// NETWORK 10
SIREN_BEACONS(ESTOP_ACTIVE := GVL_Alarms.EMERGENCY_STOP_COMMON, ERRORS_ACTIVE := APP_WARNINGS_ERRORS.ERRORS_ACTIVE, WARNINGS_ACTIVE := APP_WARNINGS_ERRORS.WARNINGS_ACTIVE);

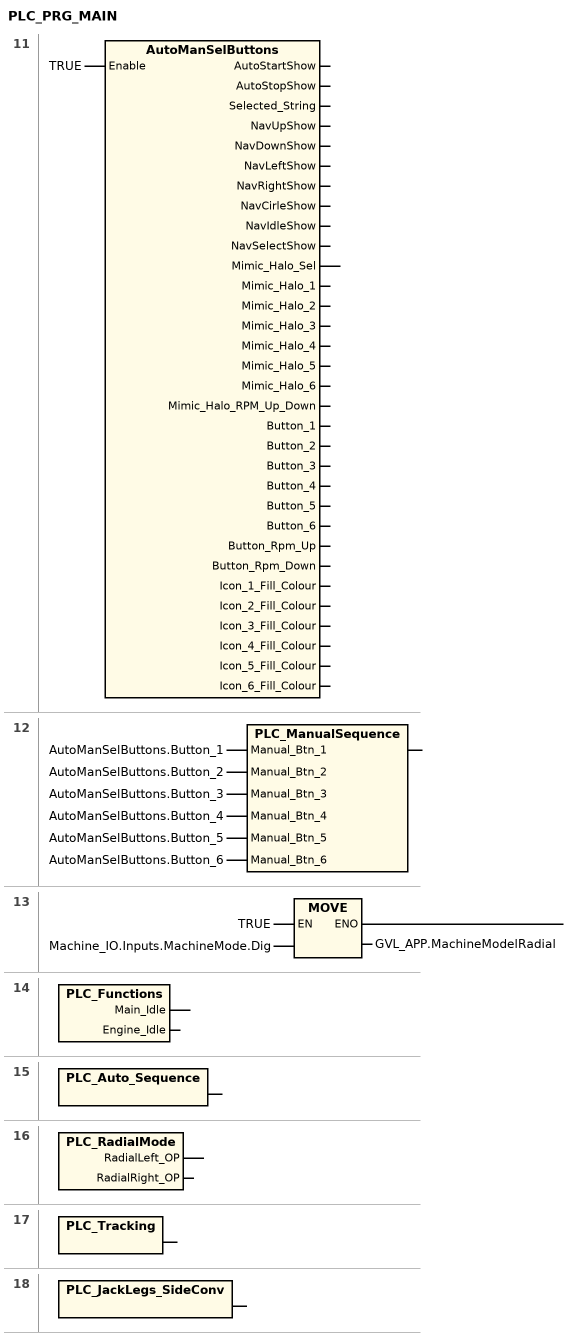
// NETWORK 11
AutoManSelButtons(Enable := TRUE);

// NETWORK 12
PLC_ManualSequence(Manual_Btn_1 := AutoManSelButtons.Button_1, Manual_Btn_2 := AutoManSelButtons.Button_2, Manual_Btn_3 := AutoManSelButtons.Button_3, Manual_Btn_4 := AutoManSelButtons.Button_4, Manual_Btn_5 := AutoManSelButtons.Button_5, Manual_Btn_6 := AutoManSelButtons.Button_6);

// NETWORK 13
GVL_APP.MachineModelRadial := Machine_IO.Inputs.MachineMode.Dig;

// NETWORK 14
PLC_Functions();

// NETWORK 15
PLC_Auto_Sequence();

// NETWORK 16
PLC_RadialMode();

// NETWORK 17
PLC_Tracking();

// NETWORK 18
PLC_JackLegs_SideConv();

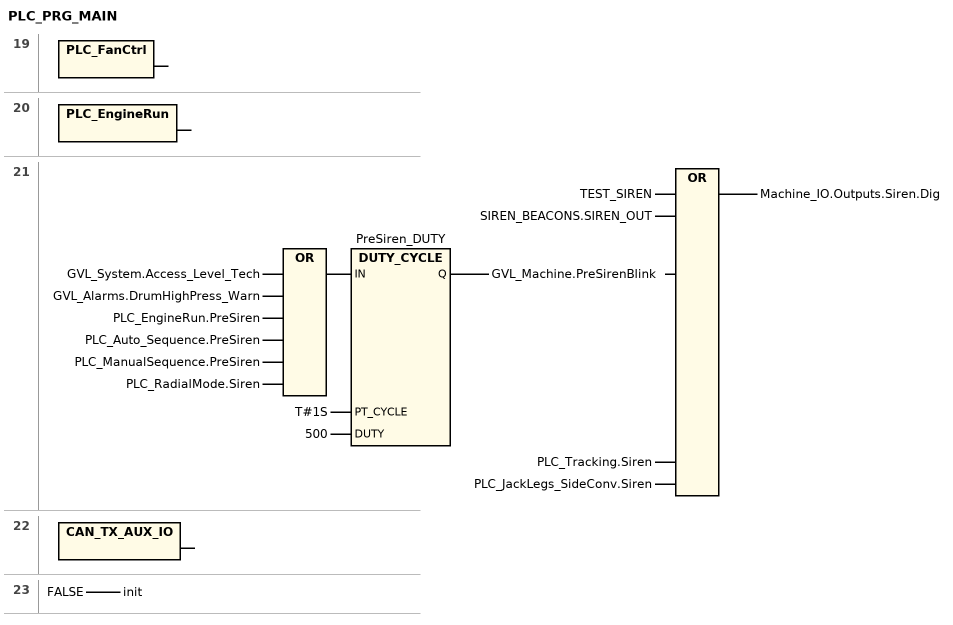
// NETWORK 19
PLC_FanCtrl();

// NETWORK 20
PLC_EngineRun();

// NETWORK 21
PreSiren_DUTY(
    IN := GVL_System.Access_Level_Tech OR GVL_Alarms.DrumHighPress_Warn OR PLC_EngineRun.PreSiren OR PLC_Auto_Sequence.PreSiren OR PLC_ManualSequence.PreSiren OR PLC_RadialMode.Siren,
    PT_CYCLE := T#1S,
    DUTY := 500); // DUTY_CYCLE
GVL_Machine.PreSirenBlink := PreSiren_DUTY.Q;
Machine_IO.Outputs.Siren.Dig := TEST_SIREN OR SIREN_BEACONS.SIREN_OUT OR PreSiren_DUTY.Q OR PLC_Tracking.Siren OR PLC_JackLegs_SideConv.Siren;

// NETWORK 22
CAN_TX_AUX_IO();

// NETWORK 23
init := FALSE;

END_PROGRAM

// Device/Application/App_PLC/PLC_SIM_MAIN
PROGRAM PLC_SIM_MAIN
VAR
END_VAR

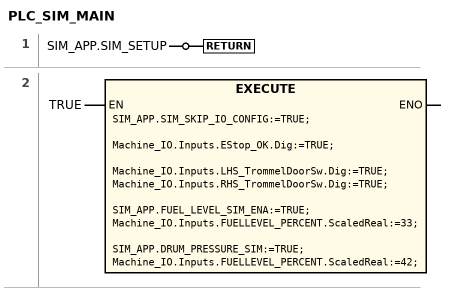
// NETWORK 1
IF NOT SIM_APP.SIM_SETUP THEN RETURN; END_IF

// NETWORK 2
SIM_APP.SIM_SKIP_IO_CONFIG:=TRUE;

Machine_IO.Inputs.EStop_OK.Dig:=TRUE;

Machine_IO.Inputs.LHS_TrommelDoorSw.Dig:=TRUE;
Machine_IO.Inputs.RHS_TrommelDoorSw.Dig:=TRUE;

SIM_APP.FUEL_LEVEL_SIM_ENA:=TRUE;
Machine_IO.Inputs.FUELLEVEL_PERCENT.ScaledReal:=33;

SIM_APP.DRUM_PRESSURE_SIM:=TRUE;
Machine_IO.Inputs.FUELLEVEL_PERCENT.ScaledReal:=42;

END_PROGRAM

// Device/Application/App_Common/System/PLC_COMMON
PROGRAM PLC_COMMON
VAR
	INIT: BOOL := TRUE;

	MAIN_HMI_Version_Info: PLC_Version_Unpack_FB;
	Version_Refresh_TON: TON;
	CHASSIS_PLC_Version_Info: SLL_IFM_Version.PLC_Version_Unpack_FB;
	
	PC_SIMULATION_MODE: INT;
	SIM_PRIME_PULSE_TON: TON;
	SIM_CAS_PRIME_PULSE_TON: TON;
	Get_Task_Info_FB: Get_Task_Info;
	TaskInfo: HMI_TASKS_INFO_STRUCT;
	SetKeyLED_FB: ifmDevice.SetKeyLED;
	
	BOOT_PIN_CODE_ENTERED: LWORD;
	BOOT_PIN_CODE_FIXED: LWORD:=2103;
	BOOT_PIN_CODE_VALID: BOOL;
	BOOT_INTO_RECOVERY: BOOL;
	BOOT_INTO_SETUP: BOOL;
	
 	BootIntoRecovery_FB: ifmDevice.BootIntoRecovery;
// 	BootIntoSetup_FB: ifmDevice.BootIntoSetup;	
 	PrintScreen_FB: ifmDevice.PrintScreen;
 	LoadSplashScreen_FB: ifmDevice.LoadSplashScreen;	
 	PrintScreenPath: STRING := '/home/cds-apps/PlcLogic/';
	SLASH_LOGO_SET: BOOL;
	HideSplashScreen_FB: ifmDevice.HideSplashScreen;
	Load_Splash_TEST: BOOL;
END_VAR

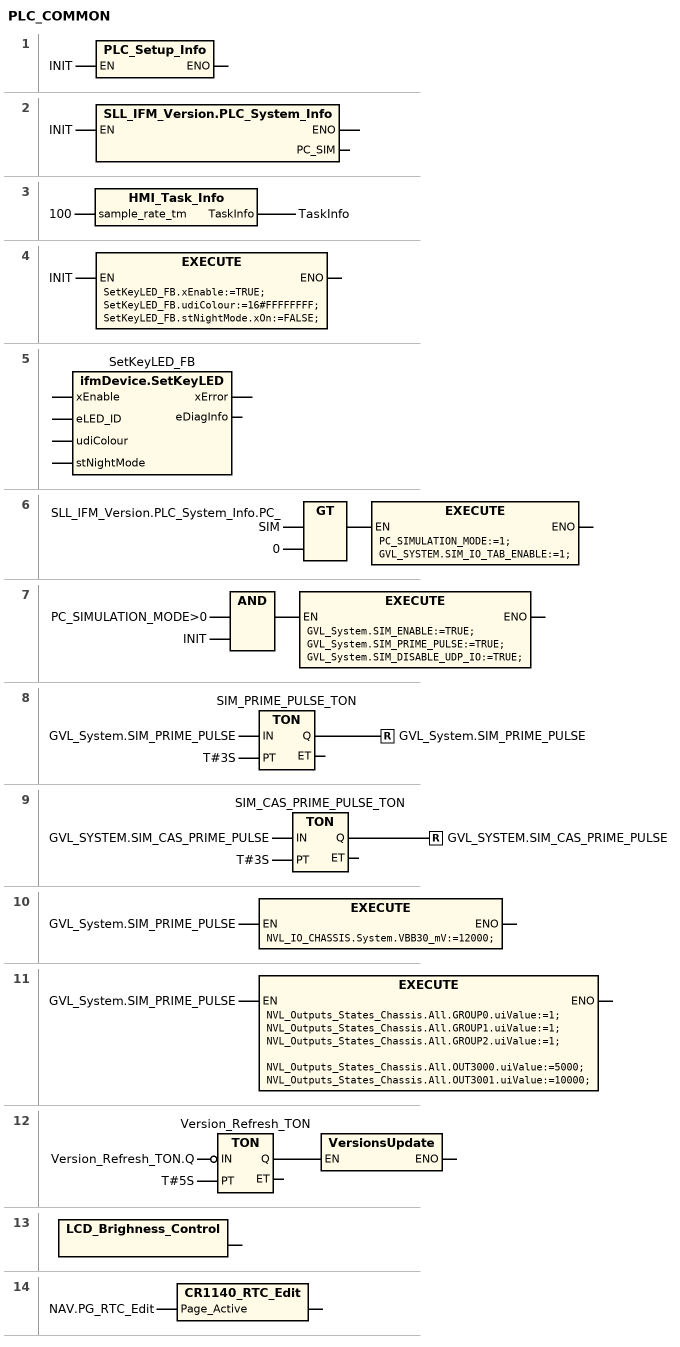
// NETWORK 1
IF INIT THEN PLC_Setup_Info(); END_IF

// NETWORK 2
IF INIT THEN SLL_IFM_Version.PLC_System_Info(); END_IF

// NETWORK 3
HMI_Task_Info(sample_rate_tm := 100);
TaskInfo := HMI_Task_Info.TaskInfo;

// NETWORK 4
IF INIT THEN
    SetKeyLED_FB.xEnable:=TRUE;
    SetKeyLED_FB.udiColour:=16#FFFFFFFF;
    SetKeyLED_FB.stNightMode.xOn:=FALSE;
END_IF

// NETWORK 5
SetKeyLED_FB(); // ifmDevice.SetKeyLED

// NETWORK 6
IF SLL_IFM_Version.PLC_System_Info.PC_SIM > 0 THEN
    PC_SIMULATION_MODE:=1;
    GVL_SYSTEM.SIM_IO_TAB_ENABLE:=1;
END_IF

// NETWORK 7
IF (PC_SIMULATION_MODE>0) AND INIT THEN
    GVL_System.SIM_ENABLE:=TRUE;
    GVL_System.SIM_PRIME_PULSE:=TRUE;
    GVL_System.SIM_DISABLE_UDP_IO:=TRUE;
END_IF

// NETWORK 8
SIM_PRIME_PULSE_TON(IN := GVL_System.SIM_PRIME_PULSE, PT := T#3S); // TON
GVL_System.SIM_PRIME_PULSE R= SIM_PRIME_PULSE_TON.Q;

// NETWORK 9
SIM_CAS_PRIME_PULSE_TON(IN := GVL_SYSTEM.SIM_CAS_PRIME_PULSE, PT := T#3S); // TON
GVL_SYSTEM.SIM_CAS_PRIME_PULSE R= SIM_CAS_PRIME_PULSE_TON.Q;

// NETWORK 10
IF GVL_System.SIM_PRIME_PULSE THEN NVL_IO_CHASSIS.System.VBB30_mV:=12000; END_IF

// NETWORK 11
IF GVL_System.SIM_PRIME_PULSE THEN
    NVL_Outputs_States_Chassis.All.GROUP0.uiValue:=1;
    NVL_Outputs_States_Chassis.All.GROUP1.uiValue:=1;
    NVL_Outputs_States_Chassis.All.GROUP2.uiValue:=1;
    
    NVL_Outputs_States_Chassis.All.OUT3000.uiValue:=5000;
    NVL_Outputs_States_Chassis.All.OUT3001.uiValue:=10000;
END_IF

// NETWORK 12
Version_Refresh_TON(IN := NOT Version_Refresh_TON.Q, PT := T#5S); // TON
IF Version_Refresh_TON.Q THEN VersionsUpdate(); END_IF

// NETWORK 13
LCD_Brighness_Control();

// NETWORK 14
CR1140_RTC_Edit(Page_Active := NAV.PG_RTC_Edit);

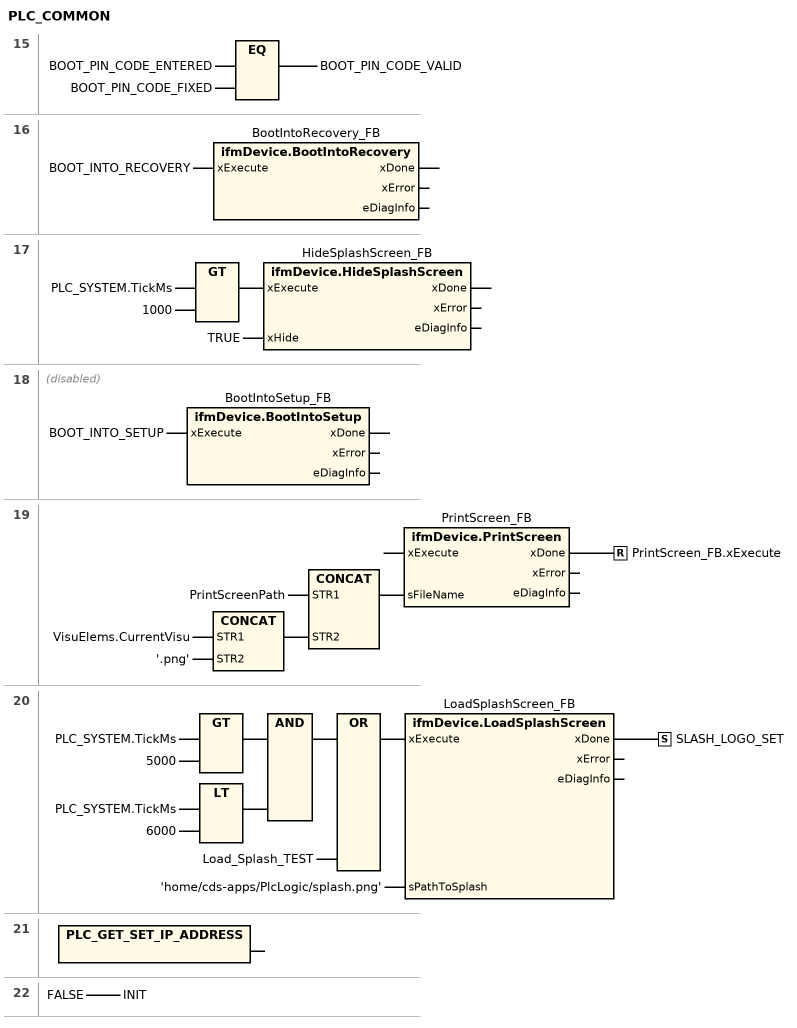
// NETWORK 15
BOOT_PIN_CODE_VALID := BOOT_PIN_CODE_ENTERED = BOOT_PIN_CODE_FIXED;

// NETWORK 16
BootIntoRecovery_FB(xExecute := BOOT_INTO_RECOVERY); // ifmDevice.BootIntoRecovery

// NETWORK 17
HideSplashScreen_FB(xExecute := PLC_SYSTEM.TickMs > 1000, xHide := TRUE); // ifmDevice.HideSplashScreen

// NETWORK 18 (disabled)
// BootIntoSetup_FB(xExecute := BOOT_INTO_SETUP); // ifmDevice.BootIntoSetup

// NETWORK 19
PrintScreen_FB(sFileName := CONCAT(STR1 := PrintScreenPath, STR2 := CONCAT(STR1 := VisuElems.CurrentVisu, STR2 := '.png'))); // ifmDevice.PrintScreen
PrintScreen_FB.xExecute R= PrintScreen_FB.xDone;

// NETWORK 20
LoadSplashScreen_FB(xExecute := PLC_SYSTEM.TickMs > 5000 AND PLC_SYSTEM.TickMs < 6000 OR Load_Splash_TEST, sPathToSplash := 'home/cds-apps/PlcLogic/splash.png'); // ifmDevice.LoadSplashScreen
SLASH_LOGO_SET S= LoadSplashScreen_FB.xDone;

// NETWORK 21
PLC_GET_SET_IP_ADDRESS();

// NETWORK 22
INIT := FALSE;

METHOD VersionsUpdate
VAR_INPUT
END_VAR
VAR
END_VAR
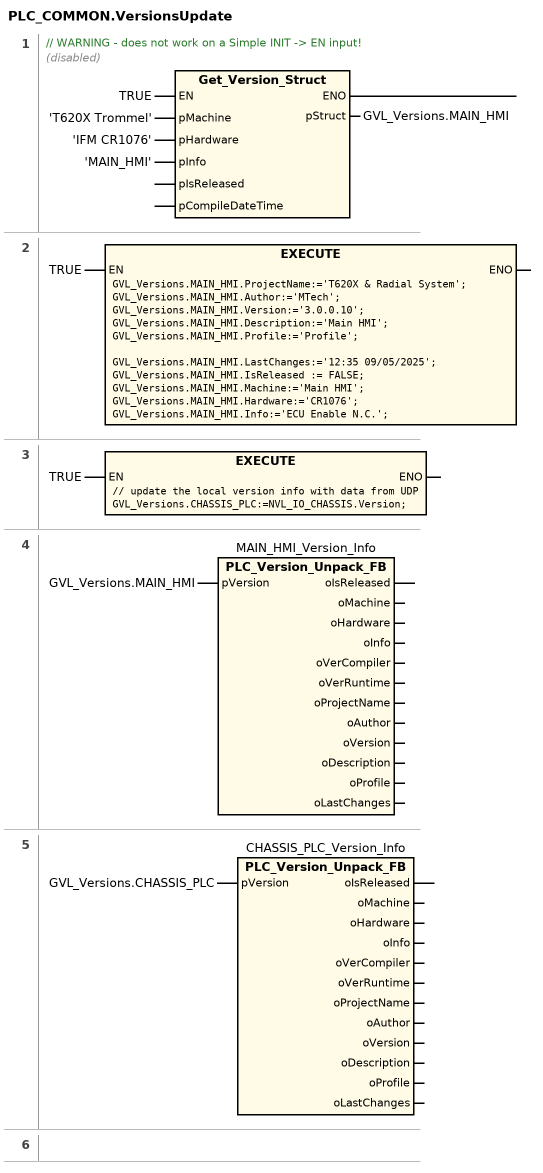
// NETWORK 1 (disabled)
// // WARNING - does not work on a Simple INIT -> EN input!
// Get_Version_Struct(pMachine := 'T620X Trommel', pHardware := 'IFM CR1076', pInfo := 'MAIN_HMI', pStruct => GVL_Versions.MAIN_HMI);

// NETWORK 2
GVL_Versions.MAIN_HMI.ProjectName:='T620X & Radial System';				
GVL_Versions.MAIN_HMI.Author:='MTech';
GVL_Versions.MAIN_HMI.Version:='3.0.0.10';
GVL_Versions.MAIN_HMI.Description:='Main HMI';
GVL_Versions.MAIN_HMI.Profile:='Profile';

GVL_Versions.MAIN_HMI.LastChanges:='12:35 09/05/2025';
GVL_Versions.MAIN_HMI.IsReleased := FALSE;
GVL_Versions.MAIN_HMI.Machine:='Main HMI';
GVL_Versions.MAIN_HMI.Hardware:='CR1076';
GVL_Versions.MAIN_HMI.Info:='ECU Enable N.C.';

// NETWORK 3
// update the local version info with data from UDP
GVL_Versions.CHASSIS_PLC:=NVL_IO_CHASSIS.Version;

// NETWORK 4
MAIN_HMI_Version_Info(pVersion := GVL_Versions.MAIN_HMI); // PLC_Version_Unpack_FB

// NETWORK 5
CHASSIS_PLC_Version_Info(pVersion := GVL_Versions.CHASSIS_PLC); // PLC_Version_Unpack_FB

// NETWORK 6
END_METHOD

END_PROGRAM

// Device/Application/App_Common/System/PLC_Setup_Info
PROGRAM PLC_Setup_Info
VAR
	INIT: BOOL:=TRUE;
END_VAR

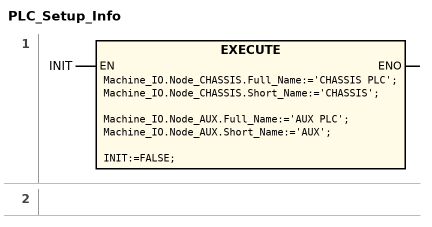
// NETWORK 1
IF INIT THEN
    Machine_IO.Node_CHASSIS.Full_Name:='CHASSIS PLC';
    Machine_IO.Node_CHASSIS.Short_Name:='CHASSIS';
    
    Machine_IO.Node_AUX.Full_Name:='AUX PLC';
    Machine_IO.Node_AUX.Short_Name:='AUX';
    
    INIT:=FALSE;
END_IF

// NETWORK 2

END_PROGRAM

// Device/Application/LIBS/HMI/HMI_Task_Info
PROGRAM HMI_Task_Info
VAR_INPUT
	sample_rate_tm:DWORD:=500;
END_VAR
VAR
	x: INT;
    hTasks:	ARRAY [0..19] OF SysTypes.RTS_IEC_HANDLE;	
    iecResult:	ARRAY [0..19] OF SysTypes.RTS_IEC_RESULT;
    sAppName:	STRING := 'Application';
    pIecInfo:	POINTER TO CmpIecTask.Task_Info2;
	last_sample_ms: DWORD;
	diff_ms: DWORD;
	finished: BOOL := FALSE;
	CpuLoadTemp: REAL;
END_VAR

VAR_OUTPUT
	TaskInfo: HMI_TASKS_INFO_STRUCT;
	CpuLoad:REAL;
END_VAR

diff_ms := SysTimeGetMs() - last_sample_ms;

IF diff_ms < sample_rate_tm THEN
	RETURN;
END_IF

x:=0;
finished:=FALSE;
CpuLoadTemp:=0;

WHILE finished = FALSE DO
	IF x = 0 THEN
		hTasks[x] := CmpIecTask.IecTaskGetFirst(pszAppName := ADR(sAppName), pResult := ADR(iecResult));
	ELSE
		hTasks[x] := IecTaskGetNext(pszAppName := ADR(sAppName), hPrevIecTask := hTasks[x-1], pResult := ADR(iecResult));
	END_IF

	IF ((hTasks[x] <> SysTypes.RTS_INVALID_HANDLE) AND (iecResult[x] = CmpErrors.Errors.ERR_OK)) THEN
		pIecInfo := CmpIecTask.IecTaskGetInfo3(hIecTask := hTasks[x],pResult := ADR(iecResult[x]));
		TaskInfo.Tasks[x].dwIntervalTask := pIecInfo^.dwInterval;
		TaskInfo.Tasks[x].dwCycleTimeTask := pIecInfo^.dwCycleTime;
		TaskInfo.Tasks[x].sNameTask := pIecInfo^.pszName^;
		TaskInfo.Tasks[x].fTaskCpuLoad:=TO_REAL(TaskInfo.Tasks[x].dwCycleTimeTask*100)/TO_REAL(TaskInfo.Tasks[x].dwIntervalTask);
		
		CpuLoadTemp:=CpuLoadTemp+TaskInfo.Tasks[x].fTaskCpuLoad;
		CpuLoad:=CpuLoadTemp;
	ELSE
		finished := TRUE;
	END_IF
	x:=x+1;
END_WHILE;

END_PROGRAM

// Device/Application/LIBS/HMI/LCD_Brighness_Control
PROGRAM LCD_Brighness_Control
VAR
	SetLCD_Backlight_FB: ifmDevice.SetLCD_Backlight;
	Brightness_Max:USINT:=100;
	Brightness_Min:USINT:=20;
	Brightness_Step:USINT:=5;
	Brightness_Key_TON: TON;	
END_VAR

VAR RETAIN
	//Brightness: USINT (0..100):=80;
END_VAR
VAR // added by the converter: edge detectors and wires of the graphical bodies
    _rt1, _rt2 : R_TRIG;
END_VAR

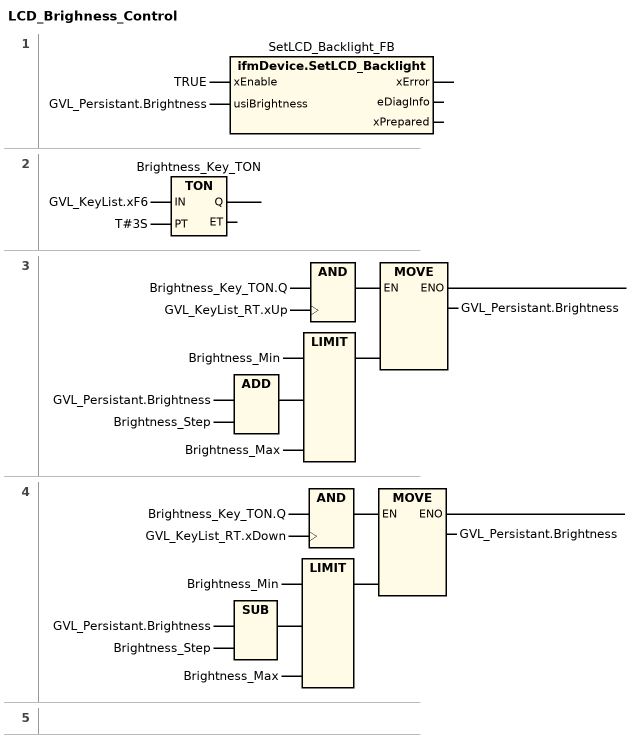
// NETWORK 1
SetLCD_Backlight_FB(xEnable := TRUE, usiBrightness := GVL_Persistant.Brightness); // ifmDevice.SetLCD_Backlight

// NETWORK 2
Brightness_Key_TON(IN := GVL_KeyList.xF6, PT := T#3S); // TON

// NETWORK 3
_rt1(CLK := GVL_KeyList_RT.xUp);
IF Brightness_Key_TON.Q AND _rt1.Q THEN
    GVL_Persistant.Brightness := LIMIT(Brightness_Min, GVL_Persistant.Brightness + Brightness_Step, Brightness_Max);
END_IF

// NETWORK 4
_rt2(CLK := GVL_KeyList_RT.xDown);
IF Brightness_Key_TON.Q AND _rt2.Q THEN
    GVL_Persistant.Brightness := LIMIT(Brightness_Min, GVL_Persistant.Brightness - Brightness_Step, Brightness_Max);
END_IF

// NETWORK 5

END_PROGRAM

// Device/Application/LIBS/HMI/CR1140_RTC_Edit
PROGRAM CR1140_RTC_Edit
VAR_INPUT
	Page_Active: BOOL;
END_VAR
VAR
	RTC_Temp: ifmDevice.stDATE_TIME;
	RTC_SetSysTime: ifmDevice.SetSysTime;
	RTC_GetSysTime: ifmDevice.GetSysTime;
	RTC_Edit_Start: BOOL;
	RTC_Edit_Done: BOOL;
	RTC_Timezone: STRING;
	RTC_GetTimeZones: ifmDevice.GetAvailableTimeZones;
	
	x: UINT;
	RTC_SetTimeZone: ifmDevice.SetTimeZone;
	ZoneSetOK: BOOL;
	TimeDateSetOK: BOOL;
	ZoneSetError: BOOL;
	TimeDateSetError: BOOL;	
	ZoneSetErrorCode: ifmTypes2.eDIAG_INFO;
	TimeDateSetErrorCode: ifmTypes2.eDIAG_INFO;	
END_VAR
VAR // added by the converter: edge detectors and wires of the graphical bodies
    _ft1, _ft2 : F_TRIG;
    _rt1, _rt2, _rt3, _rt4, _rt5, _rt6 : R_TRIG;
END_VAR

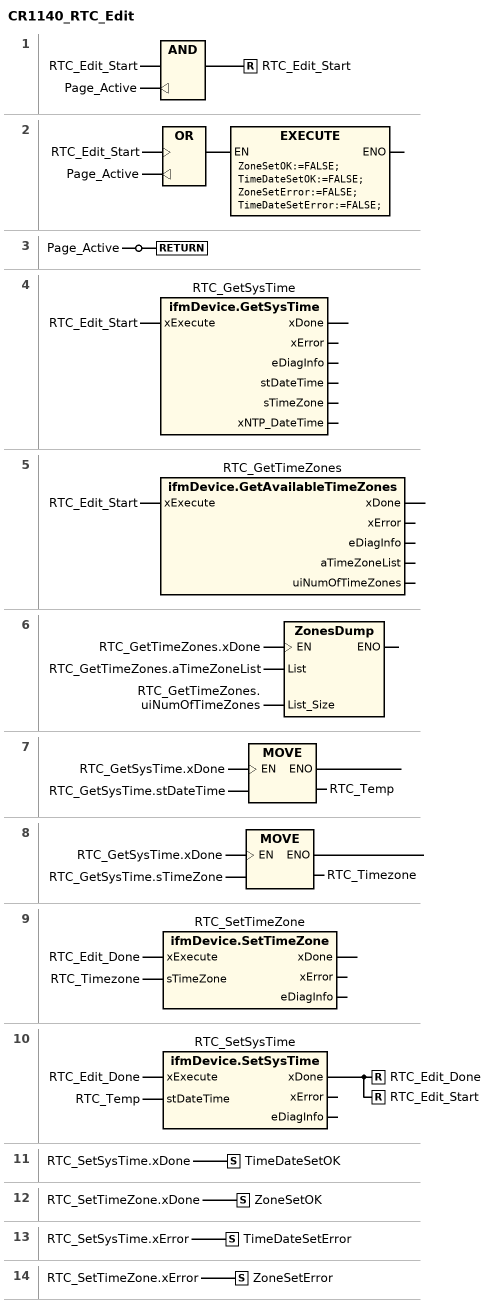
// NETWORK 1
_ft1(CLK := Page_Active);
RTC_Edit_Start R= RTC_Edit_Start AND _ft1.Q;

// NETWORK 2
_rt1(CLK := RTC_Edit_Start);
_ft2(CLK := Page_Active);
IF _rt1.Q OR _ft2.Q THEN
    ZoneSetOK:=FALSE;
    TimeDateSetOK:=FALSE;
    ZoneSetError:=FALSE;
    TimeDateSetError:=FALSE;
END_IF

// NETWORK 3
IF NOT Page_Active THEN RETURN; END_IF

// NETWORK 4
RTC_GetSysTime(xExecute := RTC_Edit_Start); // ifmDevice.GetSysTime

// NETWORK 5
RTC_GetTimeZones(xExecute := RTC_Edit_Start); // ifmDevice.GetAvailableTimeZones

// NETWORK 6
_rt2(CLK := RTC_GetTimeZones.xDone);
IF _rt2.Q THEN
    ZonesDump(List := RTC_GetTimeZones.aTimeZoneList, List_Size := RTC_GetTimeZones.uiNumOfTimeZones);
END_IF

// NETWORK 7
_rt3(CLK := RTC_GetSysTime.xDone);
IF _rt3.Q THEN RTC_Temp := RTC_GetSysTime.stDateTime; END_IF

// NETWORK 8
_rt4(CLK := RTC_GetSysTime.xDone);
IF _rt4.Q THEN RTC_Timezone := RTC_GetSysTime.sTimeZone; END_IF

// NETWORK 9
RTC_SetTimeZone(xExecute := RTC_Edit_Done, sTimeZone := RTC_Timezone); // ifmDevice.SetTimeZone

// NETWORK 10
RTC_SetSysTime(xExecute := RTC_Edit_Done, stDateTime := RTC_Temp); // ifmDevice.SetSysTime
RTC_Edit_Done R= RTC_SetSysTime.xDone;
RTC_Edit_Start R= RTC_SetSysTime.xDone;

// NETWORK 11
TimeDateSetOK S= RTC_SetSysTime.xDone;

// NETWORK 12
ZoneSetOK S= RTC_SetTimeZone.xDone;

// NETWORK 13
TimeDateSetError S= RTC_SetSysTime.xError;

// NETWORK 14
ZoneSetError S= RTC_SetTimeZone.xError;

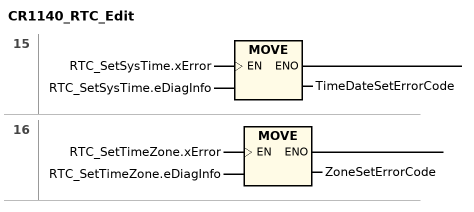
// NETWORK 15
_rt5(CLK := RTC_SetSysTime.xError);
IF _rt5.Q THEN TimeDateSetErrorCode := RTC_SetSysTime.eDiagInfo; END_IF

// NETWORK 16
_rt6(CLK := RTC_SetTimeZone.xError);
IF _rt6.Q THEN ZoneSetErrorCode := RTC_SetTimeZone.eDiagInfo; END_IF

METHOD ZonesDump
VAR_INPUT
	List: REFERENCE TO ifmDevice.aTIME_ZONE_LIST;
	List_Size: UINT;
END_VAR
VAR
	g_sMainDirectory : STRING := 'App'; // Base directory can be adapted. NOTE: Since V3.5.19.0 file access to an absolute path is denied normally.
	szFileName  		: STRING(128);
	
	hFile        	: RTS_IEC_HANDLE := RTS_INVALID_HANDLE;
	udiPos			: __XWORD;
	udiWrite		: __XWORD;
	
	(* Error Codes *)
	udiPosError	 		: RTS_IEC_RESULT;
	udiDeleteError		: RTS_IEC_RESULT;
	udiWriteError		: RTS_IEC_RESULT;
	udiOpenError		: RTS_IEC_RESULT;
	udiCloseError		: RTS_IEC_RESULT;
	
	X:UINT;
	TempString: STRING;
	
// 	CheckDir:BOOL;
// 	udiResult		: __XWORD;
// 	udiReadError: UDINT;	
// 	udiDirHandle	: RTS_IEC_HANDLE;
// 	udiFileHandle	: RTS_IEC_HANDLE;		
// 	sDirEntry		: STRING(1024);	
// 	stDirInfo		: DirInfo;
// 	iFilesCount		: INT;	
END_VAR
//In the following the file access with the SysFile library is shown

(* At the beginning a file is opened and a string is written into that file.
   After the modification of the file it must be closed.
   The access modifier AM_WRITE_PLUS is used. All modifiers with "_PLUS" have read/write access.
   However the function SysFileGetPos must be used to get an valid pointer position for writing. *)
	(* The file names can be adapted *)

szFileName := CONCAT(g_sMainDirectory, '/ZoneDump.txt');		

(* delete existing example files*)
udiDeleteError:=SysFileDelete(szFileName:=szFileName );

// IF CheckDir THEN
// 	(* open the directory 
// 		the handle is returned and the first directory entry. Normally the first entry is "." and the second ".."*)
// 	udiDirHandle := SysDirOpen(szDir:= g_sMainDirectory, szDirEntry:= sDirEntry, diMaxDirEntry:= SIZEOF(sDirEntry), 
// 				pDirInfo:= ADR(stDirInfo), pResult:= udiResult);
// 	
// 	(* Iterate through all direcotry entries and count them. The implicit entries with points are not count.
// 		when the last entry is reached the SysDirRead always delivers the last entry.*)
// 	iFilesCount := 0;
// 	IF udiResult = CmpErrors.Errors.ERR_OK AND udiFileHandle <> RTS_INVALID_HANDLE THEN
// 		REPEAT
// 			IF FIND(sDirEntry, '.') <> 1  THEN
// 				iFilesCount := iFilesCount +1;
// 			END_IF
// 			udiReadError:= SysDirRead(hDir:= udiDirHandle, szDirEntry:= sDirEntry, diMaxDirEntry:= SIZEOF(sDirEntry), pDirInfo:=ADR(stDirInfo) );
// 		UNTIL
// 			udiReadError = CmpErrors.Errors.ERR_END_OF_OBJECT
// 		END_REPEAT
// 	END_IF	
// 
// 	(* Close the directory *)
// 	udiCloseError := SysDirClose(hDir:= udiDirHandle);	
// END_IF

hFile := SysFileOpen(szFile:=szFileName, am:=SysFile.AM_WRITE_PLUS, pResult:=ADR(udiOpenError));
IF hFile <> RTS_INVALID_HANDLE	THEN
	udiPosError := SysFileGetPos(hFile:=hFile, pulPos:=ADR(udiPos));
	
	FOR x := 0 TO List_Size DO
		TempString:=TO_STRING(x);
		TempString:=CONCAT(TempString,',');	
		TempString:=CONCAT(TempString,List[x]);	
		TempString:=CONCAT(TempString,'$0d');
		udiWrite := SysFileWrite(hFile:=hFile, pbyBuffer:=ADR(TempString), ulSize:=INT_TO_UDINT(LEN(TempString)), pResult:=ADR(udiWriteError));
	END_FOR

	udiCloseError  := SysFileClose(hFile:=hFile);
END_IF
END_METHOD

END_PROGRAM

// Device/Application/App_Common/Nav/Nav
PROGRAM Nav
VAR	
	INIT: BOOL:=TRUE;
	
	NAV_RIGHT_PAGE_COM: BOOL;
	NAV_LEFT_PAGE_COM: BOOL;
	
	DEFAULT_HOME_PAGE: STRING;
	
	RETURN_STACK: ARRAY[0..4] OF STRING;
	
	VIZNAME_Prefix: STRING:='Visualization_';	
	VIZNAME_MAIN_1: STRING:= 'Visualization_Main_1';
	VIZNAME_MANUAL_1: STRING:= 'Visualization_Manual_1';
	VIZNAME_MANUAL_2: STRING:= 'Visualization_Manual_2';	
	VIZNAME_ENGINE_1: STRING:= 'Visualization_Engine_1';
	VIZNAME_ENGINE_2: STRING:= 'Visualization_Engine_2';		
	VIZNAME_SETTINGS_RTC: STRING:='Visualization_Settings_RTC';
	VIZNAME_LOG_MAIN: STRING:='Visualization_Settings_IO_Log';
																
	VISNAME_SECURITY_QRCODE_LOGIN: STRING:='Visualization_Security_QRcode_Login';
	
	VIZNAME_DIAG_NAMES_PAGES: ARRAY [0..19] OF STRING[40]:=[	
															'Default',
															'Text input',
															'Text input with limits',
															'VisuDialogs.Keypad',
															'VisuDialogs.Numpad',
															'VisuDialogs.NumpadExtended',
															'VisuDialogs_Template.Keypad',
															'VisuDialogs_Template.Numpad',
															'VisuDialogs_Template.NumpadExtended',
															'VisuDialogs_Template.TextinputWithLimits',
															'Output_Force',
															'VisuDialogs.FileOpenSave',
															'VisuDialogs.Login',
															'VisuDialogs.MessageBox',
															'VisuDialogs_Template.FileOpenSave',
															'VisuDialogs_Template.Login',
															'VisuDialogs_Template.MessageBox',															
															''];		
	
	VIZNAME_SETTINGS_PAGES: ARRAY [0..19] OF STRING[40]:=[	'Visualization_Settings_Main', 		// 0
															'Visualization_Net_Status',			// 1
															'Visualization_PLC_Versions',		// 2														
															'Visualization_Settings_Misc',		// 3
															'Visualization_Settings_RTC',		// 4
															'Visualization_Net_Status_Adv',		// 5
															'Visualization_PLC_Status',			// 6																							
															'Visualization_Settings_IO_Log',	// 7
															''];															

	VIZNAME_APP_SETTINGS_PAGES: ARRAY [0..19] OF STRING[40]:=[	'Visualization_Settings_1', 		// 0
															'Visualization_Settings_2',			// 1
															'Visualization_Settings_3',		// 2		
															'Visualization_Settings_4',		// 3		
															''];	// 7

	VIZNAME_ALARMS_PAGES: ARRAY [0..19] OF STRING[40]:=[	'Visualization_Alarms_Main',
															'Visualization_Alarms_IO',
															'Visualization_Alarms_Hist',
															''];															

	VIZNAME_ENGINE_PAGES: ARRAY [0..19] OF STRING[40]:=[	'Visualization_Engine_1',
															'Visualization_Engine_2',
															'Visualization_Engine_3',															
															''];
	
	VIZNAME_DIAG_IO_PAGES: ARRAY [0..19] OF STRING[40]:=[	
															'Visualization_DIAG_IO_Ip_G0',
															'Visualization_DIAG_IO_Ip_G1',
															'Visualization_DIAG_IO_Ip_G2',												
															'Visualization_DIAG_IO_Op_G0',
															'Visualization_DIAG_IO_Op_G1',
															'Visualization_DIAG_IO_Op_G2',
															'Visualization_DIAG_IO_AUX',															
															''];															
																											

	PG_SETTINGS_MAIN: BOOL;
	PG_ALARMS_MAIN: BOOL;
	PG_ALARMS_IO: BOOL;	
	PG_ALARMS_HIST: BOOL;
	PG_MAIN_1: BOOL;
	PG_MANUAL_1: BOOL;
	PG_MANUAL_2: BOOL;
	PG_RTC_Edit: BOOL;
	PG_LOG_MAIN: BOOL;	
	
	PG_ENGINE_1: BOOL;
	PG_ENGINE_2: BOOL;	
	
	PG_APP_SETTINGS_1: BOOL;
	PG_APP_SETTINGS_2: BOOL;
	PG_APP_SETTINGS_3: BOOL;	
	
	NAV_TO_SETTINGS: BOOL;
	NAV_TO_IO_DIAG_PAGES: BOOL;
	
	Access_Tech_Level: BOOL;
	
	Nav_Pages_Group_Settings_FB: Nav_Pages_Group_FB;
	Nav_Pages_Group_App_Settings_FB: Nav_Pages_Group_FB;
	Nav_Pages_Group_Main_FB: Nav_Pages_Group_FB;
	Nav_Pages_Group_IO_Diag_FB: Nav_Pages_Group_FB;
	Nav_Pages_Group_Alarms_FB: Nav_Pages_Group_FB;
	Nav_Pages_Group_ENGINE_FB: Nav_Pages_Group_FB;
	
	Head_PageName: STRING;
	
	NAV_NODE_UNAVAIL_DUTY_CYCLE: DUTY_CYCLE;
	KEYS_ACTIVE: BOOL;
	KEYS_INACTIVE_TON: TON;
	KEYS_INACTIVE_TM: TIME;
	CAS_SCREEN_DUTY_CYCLE: DUTY_CYCLE;
	
	Footer_ShowDiagSwitch: BOOL;
	Footer_ShowNavLeft:BOOL;
	Footer_ShowNavRight:BOOL;
	Footer_ShowAlmAck:BOOL;	
	
	AckAll_TON: TON;
	AckAll_TP: TP;
	
	Alarms_Main_Selected_Row: INT;
	Alarms_IO_Selected_Row: INT;
	Alarms_Hist_Selected_Row: INT;
	
	Alarms_Main_Count: INT;
	Alarms_IO_Count: INT;
	Alarms_Hist_Count: INT;
	Alarms_Hist_Count_Prev: INT;
	
	PG_ALARMS_MAIN_CLEAR_ALL_TON: TON;
	PG_ALARMS_MAIN_CLEAR_INACTIVE_TON: TON;
	DIAGS_OPEN: BOOL;
	FORCE_HOME_TON: TON;
	FALS: BOOL;
	LED_Control_Diags_FB: LED_Control_FB;
	LED_Control_Main_1_FB: LED_Control_FB;
	LED_Control_Settings_Main_FB: LED_Control_FB;
	LED_Control_Main_1_TON: TON;
	LED_Control_Settings_Main_TON: TON;
	LED_Control_Diags_TON: TON;
END_VAR
VAR // added by the converter: edge detectors and wires of the graphical bodies
    _w1, _w2 : BOOL;
    _rt1, _rt2, _rt3, _rt4, _rt5, _rt6, _rt7, _rt8, _rt9, _rt10, _rt11, _rt12, _rt13, _rt14 : R_TRIG;
    _ft1 : F_TRIG;
END_VAR

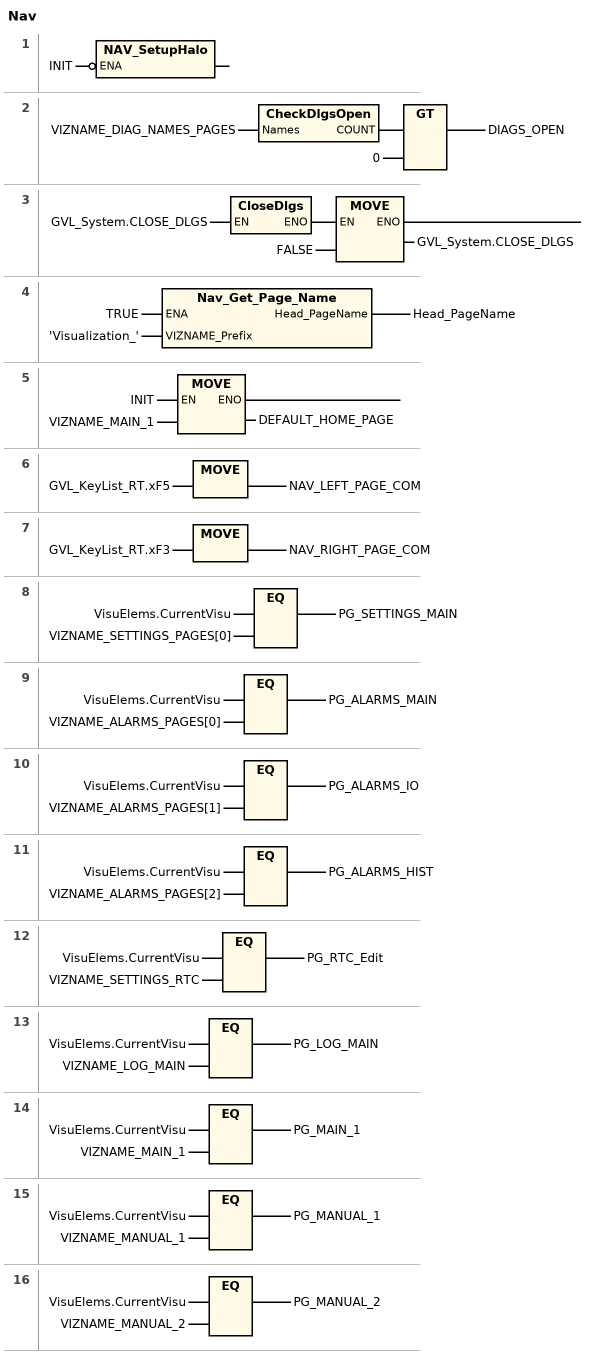
// NETWORK 1
NAV_SetupHalo(ENA := NOT INIT);

// NETWORK 2
CheckDlgsOpen(Names := VIZNAME_DIAG_NAMES_PAGES);
DIAGS_OPEN := CheckDlgsOpen.COUNT > 0;

// NETWORK 3
_w1 := GVL_System.CLOSE_DLGS;
IF _w1 THEN CloseDlgs(); END_IF
IF _w1 THEN GVL_System.CLOSE_DLGS := FALSE; END_IF

// NETWORK 4
Nav_Get_Page_Name(ENA := TRUE, VIZNAME_Prefix := 'Visualization_');
Head_PageName := Nav_Get_Page_Name.Head_PageName;

// NETWORK 5
IF INIT THEN DEFAULT_HOME_PAGE := VIZNAME_MAIN_1; END_IF

// NETWORK 6
NAV_LEFT_PAGE_COM := GVL_KeyList_RT.xF5;

// NETWORK 7
NAV_RIGHT_PAGE_COM := GVL_KeyList_RT.xF3;

// NETWORK 8
PG_SETTINGS_MAIN := VisuElems.CurrentVisu = VIZNAME_SETTINGS_PAGES[0];

// NETWORK 9
PG_ALARMS_MAIN := VisuElems.CurrentVisu = VIZNAME_ALARMS_PAGES[0];

// NETWORK 10
PG_ALARMS_IO := VisuElems.CurrentVisu = VIZNAME_ALARMS_PAGES[1];

// NETWORK 11
PG_ALARMS_HIST := VisuElems.CurrentVisu = VIZNAME_ALARMS_PAGES[2];

// NETWORK 12
PG_RTC_Edit := VisuElems.CurrentVisu = VIZNAME_SETTINGS_RTC;

// NETWORK 13
PG_LOG_MAIN := VisuElems.CurrentVisu = VIZNAME_LOG_MAIN;

// NETWORK 14
PG_MAIN_1 := VisuElems.CurrentVisu = VIZNAME_MAIN_1;

// NETWORK 15
PG_MANUAL_1 := VisuElems.CurrentVisu = VIZNAME_MANUAL_1;

// NETWORK 16
PG_MANUAL_2 := VisuElems.CurrentVisu = VIZNAME_MANUAL_2;

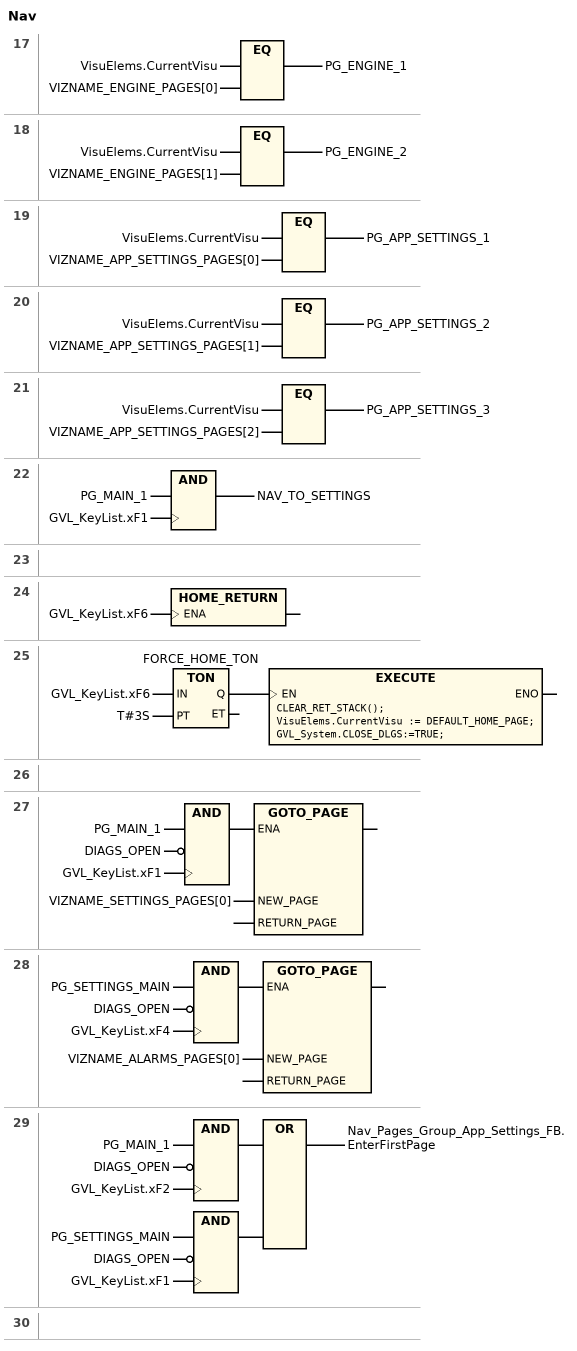
// NETWORK 17
PG_ENGINE_1 := VisuElems.CurrentVisu = VIZNAME_ENGINE_PAGES[0];

// NETWORK 18
PG_ENGINE_2 := VisuElems.CurrentVisu = VIZNAME_ENGINE_PAGES[1];

// NETWORK 19
PG_APP_SETTINGS_1 := VisuElems.CurrentVisu = VIZNAME_APP_SETTINGS_PAGES[0];

// NETWORK 20
PG_APP_SETTINGS_2 := VisuElems.CurrentVisu = VIZNAME_APP_SETTINGS_PAGES[1];

// NETWORK 21
PG_APP_SETTINGS_3 := VisuElems.CurrentVisu = VIZNAME_APP_SETTINGS_PAGES[2];

// NETWORK 22
_rt1(CLK := GVL_KeyList.xF1);
NAV_TO_SETTINGS := PG_MAIN_1 AND _rt1.Q;

// NETWORK 23

// NETWORK 24
_rt2(CLK := GVL_KeyList.xF6);
HOME_RETURN(ENA := _rt2.Q);

// NETWORK 25
FORCE_HOME_TON(IN := GVL_KeyList.xF6, PT := T#3S); // TON
_rt3(CLK := FORCE_HOME_TON.Q);
IF _rt3.Q THEN
    CLEAR_RET_STACK();
    VisuElems.CurrentVisu := DEFAULT_HOME_PAGE;
    GVL_System.CLOSE_DLGS:=TRUE;
END_IF

// NETWORK 26

// NETWORK 27
_rt4(CLK := GVL_KeyList.xF1);
GOTO_PAGE(ENA := PG_MAIN_1 AND NOT DIAGS_OPEN AND _rt4.Q, NEW_PAGE := VIZNAME_SETTINGS_PAGES[0]);

// NETWORK 28
_rt5(CLK := GVL_KeyList.xF4);
GOTO_PAGE(ENA := PG_SETTINGS_MAIN AND NOT DIAGS_OPEN AND _rt5.Q, NEW_PAGE := VIZNAME_ALARMS_PAGES[0]);

// NETWORK 29
_rt6(CLK := GVL_KeyList.xF2);
_rt7(CLK := GVL_KeyList.xF1);
Nav_Pages_Group_App_Settings_FB.EnterFirstPage := PG_MAIN_1 AND NOT DIAGS_OPEN AND _rt6.Q OR PG_SETTINGS_MAIN AND NOT DIAGS_OPEN AND _rt7.Q;

// NETWORK 30

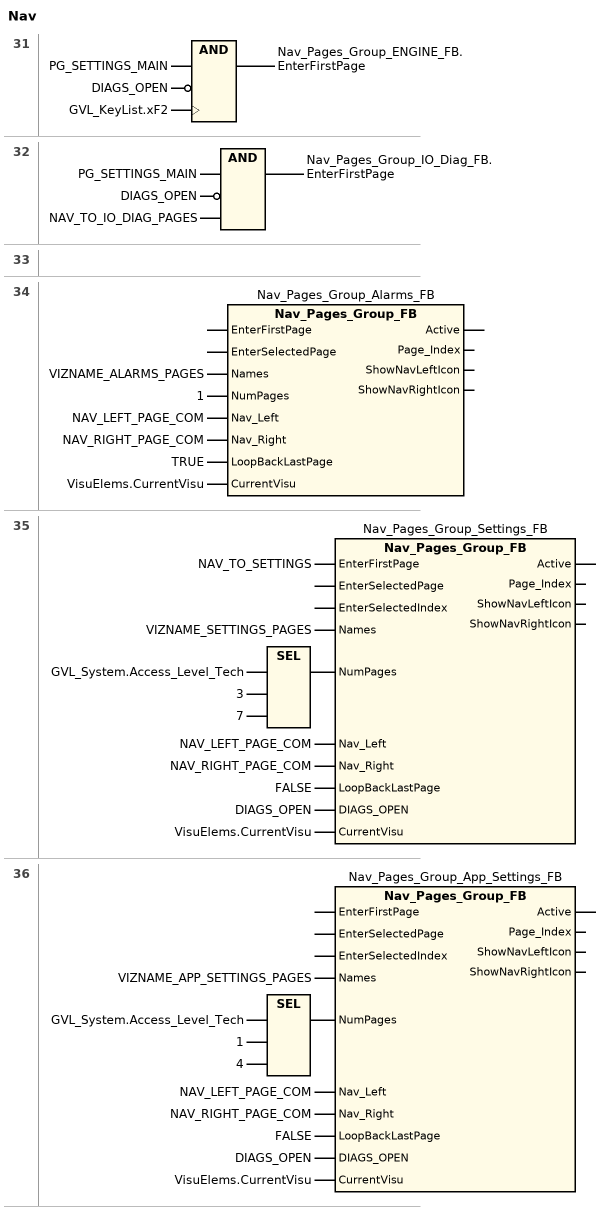
// NETWORK 31
_rt8(CLK := GVL_KeyList.xF2);
Nav_Pages_Group_ENGINE_FB.EnterFirstPage := PG_SETTINGS_MAIN AND NOT DIAGS_OPEN AND _rt8.Q;

// NETWORK 32
Nav_Pages_Group_IO_Diag_FB.EnterFirstPage := PG_SETTINGS_MAIN AND NOT DIAGS_OPEN AND NAV_TO_IO_DIAG_PAGES;

// NETWORK 33

// NETWORK 34
Nav_Pages_Group_Alarms_FB(
    Names := VIZNAME_ALARMS_PAGES,
    NumPages := 1,
    Nav_Left := NAV_LEFT_PAGE_COM,
    Nav_Right := NAV_RIGHT_PAGE_COM,
    LoopBackLastPage := TRUE,
    CurrentVisu := VisuElems.CurrentVisu); // Nav_Pages_Group_FB

// NETWORK 35
Nav_Pages_Group_Settings_FB(
    EnterFirstPage := NAV_TO_SETTINGS,
    Names := VIZNAME_SETTINGS_PAGES,
    NumPages := SEL(GVL_System.Access_Level_Tech, 3, 7),
    Nav_Left := NAV_LEFT_PAGE_COM,
    Nav_Right := NAV_RIGHT_PAGE_COM,
    LoopBackLastPage := FALSE,
    DIAGS_OPEN := DIAGS_OPEN,
    CurrentVisu := VisuElems.CurrentVisu); // Nav_Pages_Group_FB

// NETWORK 36
Nav_Pages_Group_App_Settings_FB(
    Names := VIZNAME_APP_SETTINGS_PAGES,
    NumPages := SEL(GVL_System.Access_Level_Tech, 1, 4),
    Nav_Left := NAV_LEFT_PAGE_COM,
    Nav_Right := NAV_RIGHT_PAGE_COM,
    LoopBackLastPage := FALSE,
    DIAGS_OPEN := DIAGS_OPEN,
    CurrentVisu := VisuElems.CurrentVisu); // Nav_Pages_Group_FB

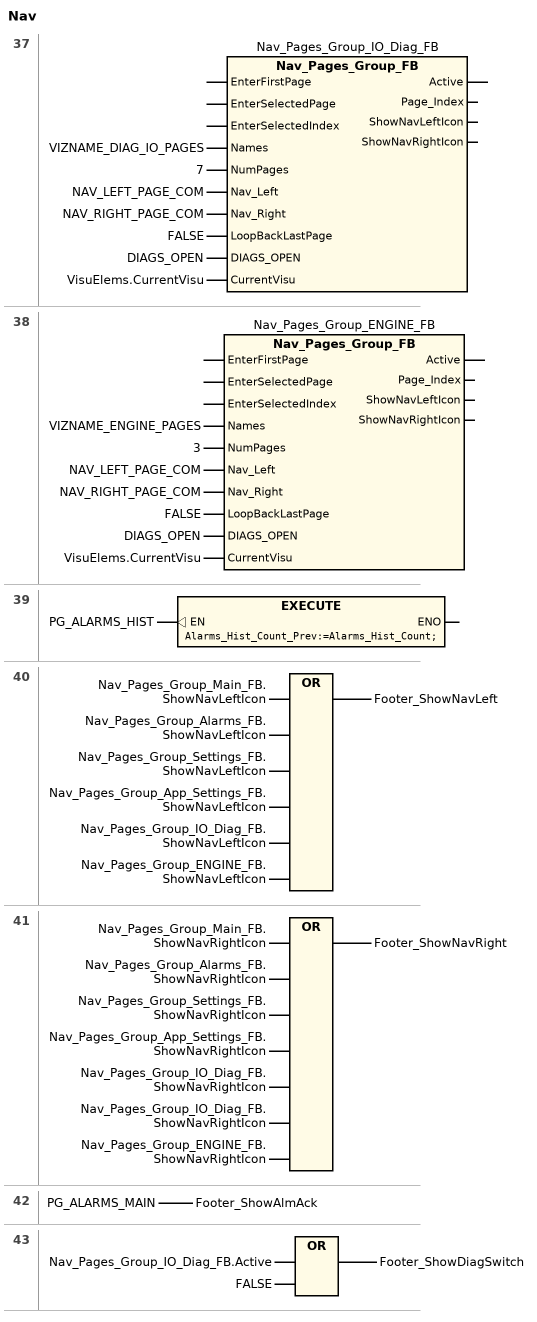
// NETWORK 37
Nav_Pages_Group_IO_Diag_FB(
    Names := VIZNAME_DIAG_IO_PAGES,
    NumPages := 7,
    Nav_Left := NAV_LEFT_PAGE_COM,
    Nav_Right := NAV_RIGHT_PAGE_COM,
    LoopBackLastPage := FALSE,
    DIAGS_OPEN := DIAGS_OPEN,
    CurrentVisu := VisuElems.CurrentVisu); // Nav_Pages_Group_FB

// NETWORK 38
Nav_Pages_Group_ENGINE_FB(
    Names := VIZNAME_ENGINE_PAGES,
    NumPages := 3,
    Nav_Left := NAV_LEFT_PAGE_COM,
    Nav_Right := NAV_RIGHT_PAGE_COM,
    LoopBackLastPage := FALSE,
    DIAGS_OPEN := DIAGS_OPEN,
    CurrentVisu := VisuElems.CurrentVisu); // Nav_Pages_Group_FB

// NETWORK 39
_ft1(CLK := PG_ALARMS_HIST);
IF _ft1.Q THEN Alarms_Hist_Count_Prev:=Alarms_Hist_Count; END_IF

// NETWORK 40
Footer_ShowNavLeft := Nav_Pages_Group_Main_FB.ShowNavLeftIcon OR Nav_Pages_Group_Alarms_FB.ShowNavLeftIcon OR Nav_Pages_Group_Settings_FB.ShowNavLeftIcon OR Nav_Pages_Group_App_Settings_FB.ShowNavLeftIcon OR Nav_Pages_Group_IO_Diag_FB.ShowNavLeftIcon OR Nav_Pages_Group_ENGINE_FB.ShowNavLeftIcon;

// NETWORK 41
Footer_ShowNavRight := Nav_Pages_Group_Main_FB.ShowNavRightIcon OR Nav_Pages_Group_Alarms_FB.ShowNavRightIcon OR Nav_Pages_Group_Settings_FB.ShowNavRightIcon OR Nav_Pages_Group_App_Settings_FB.ShowNavRightIcon OR Nav_Pages_Group_IO_Diag_FB.ShowNavRightIcon OR Nav_Pages_Group_IO_Diag_FB.ShowNavRightIcon OR Nav_Pages_Group_ENGINE_FB.ShowNavRightIcon;

// NETWORK 42
Footer_ShowAlmAck := PG_ALARMS_MAIN;

// NETWORK 43
Footer_ShowDiagSwitch := Nav_Pages_Group_IO_Diag_FB.Active OR FALSE;

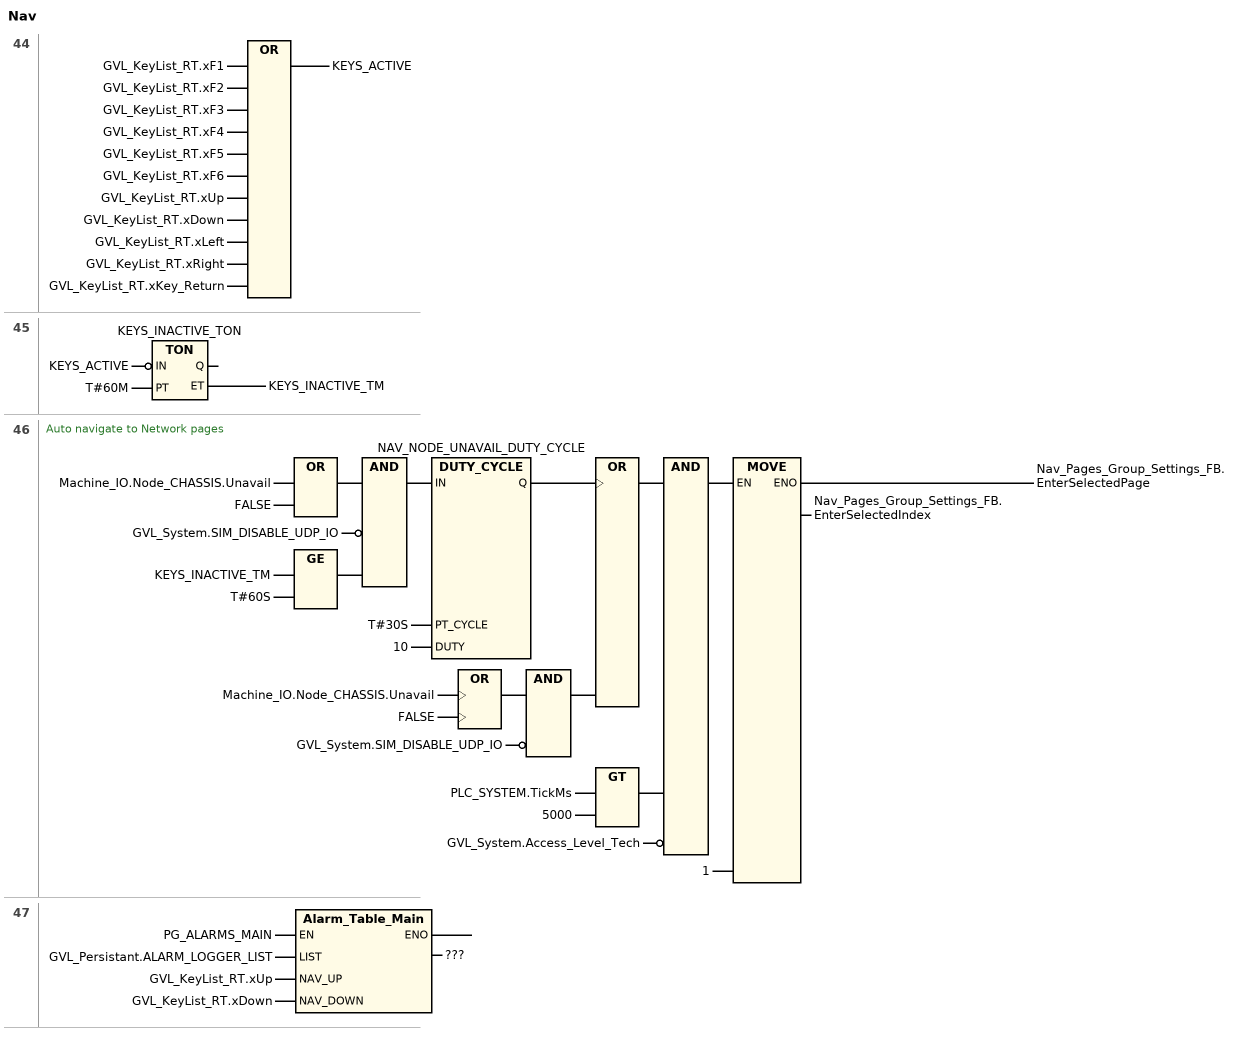
// NETWORK 44
KEYS_ACTIVE := GVL_KeyList_RT.xF1 OR GVL_KeyList_RT.xF2 OR GVL_KeyList_RT.xF3 OR GVL_KeyList_RT.xF4 OR GVL_KeyList_RT.xF5 OR GVL_KeyList_RT.xF6 OR GVL_KeyList_RT.xUp OR GVL_KeyList_RT.xDown OR GVL_KeyList_RT.xLeft OR GVL_KeyList_RT.xRight OR GVL_KeyList_RT.xKey_Return;

// NETWORK 45
KEYS_INACTIVE_TON(IN := NOT KEYS_ACTIVE, PT := T#60M); // TON
KEYS_INACTIVE_TM := KEYS_INACTIVE_TON.ET;

// NETWORK 46
// Auto navigate to Network pages
NAV_NODE_UNAVAIL_DUTY_CYCLE(
    IN := (Machine_IO.Node_CHASSIS.Unavail OR FALSE) AND NOT GVL_System.SIM_DISABLE_UDP_IO AND KEYS_INACTIVE_TM >= T#60S,
    PT_CYCLE := T#30S,
    DUTY := 10); // DUTY_CYCLE
_rt9(CLK := NAV_NODE_UNAVAIL_DUTY_CYCLE.Q);
_rt10(CLK := Machine_IO.Node_CHASSIS.Unavail);
_rt11(CLK := FALSE);
_w2 := (_rt9.Q OR (_rt10.Q OR _rt11.Q) AND NOT GVL_System.SIM_DISABLE_UDP_IO) AND PLC_SYSTEM.TickMs > 5000 AND NOT GVL_System.Access_Level_Tech;
IF _w2 THEN Nav_Pages_Group_Settings_FB.EnterSelectedIndex := 1; END_IF
Nav_Pages_Group_Settings_FB.EnterSelectedPage := _w2;

// NETWORK 47
IF PG_ALARMS_MAIN THEN
    Alarm_Table_Main(LIST := GVL_Persistant.ALARM_LOGGER_LIST, NAV_UP := GVL_KeyList_RT.xUp, NAV_DOWN := GVL_KeyList_RT.xDown);
END_IF

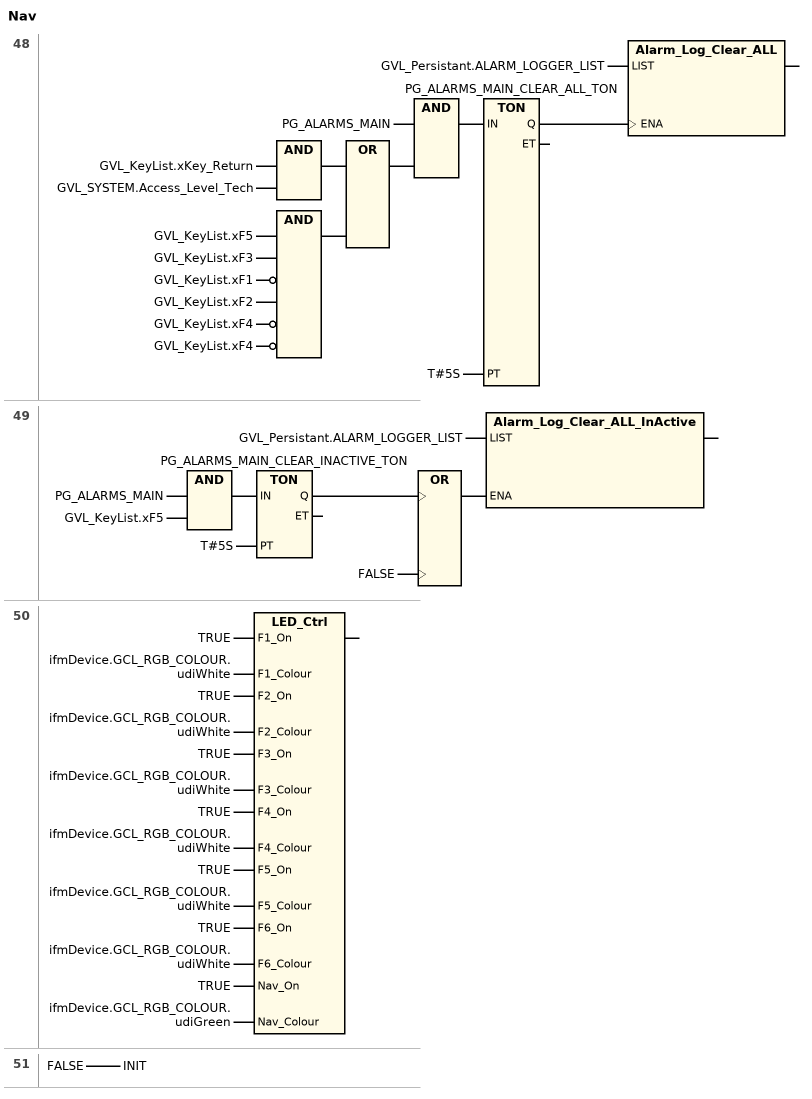
// NETWORK 48
PG_ALARMS_MAIN_CLEAR_ALL_TON(IN := PG_ALARMS_MAIN AND (GVL_KeyList.xKey_Return AND GVL_SYSTEM.Access_Level_Tech OR GVL_KeyList.xF5 AND GVL_KeyList.xF3 AND NOT GVL_KeyList.xF1 AND GVL_KeyList.xF2 AND NOT GVL_KeyList.xF4 AND NOT GVL_KeyList.xF4), PT := T#5S); // TON
_rt12(CLK := PG_ALARMS_MAIN_CLEAR_ALL_TON.Q);
Alarm_Log_Clear_ALL(LIST := GVL_Persistant.ALARM_LOGGER_LIST, ENA := _rt12.Q);

// NETWORK 49
PG_ALARMS_MAIN_CLEAR_INACTIVE_TON(IN := PG_ALARMS_MAIN AND GVL_KeyList.xF5, PT := T#5S); // TON
_rt13(CLK := PG_ALARMS_MAIN_CLEAR_INACTIVE_TON.Q);
_rt14(CLK := FALSE);
Alarm_Log_Clear_ALL_InActive(LIST := GVL_Persistant.ALARM_LOGGER_LIST, ENA := _rt13.Q OR _rt14.Q);

// NETWORK 50
LED_Ctrl(F1_On := TRUE, F1_Colour := ifmDevice.GCL_RGB_COLOUR.udiWhite, F2_On := TRUE, F2_Colour := ifmDevice.GCL_RGB_COLOUR.udiWhite, F3_On := TRUE, F3_Colour := ifmDevice.GCL_RGB_COLOUR.udiWhite, F4_On := TRUE, F4_Colour := ifmDevice.GCL_RGB_COLOUR.udiWhite, F5_On := TRUE, F5_Colour := ifmDevice.GCL_RGB_COLOUR.udiWhite, F6_On := TRUE, F6_Colour := ifmDevice.GCL_RGB_COLOUR.udiWhite, Nav_On := TRUE, Nav_Colour := ifmDevice.GCL_RGB_COLOUR.udiGreen);

// NETWORK 51
INIT := FALSE;

METHOD CLEAR_RET_STACK : STRING
VAR_INPUT
END_VAR
RETURN_STACK[0]:='';
RETURN_STACK[1]:='';
RETURN_STACK[2]:='';
RETURN_STACK[3]:='';
RETURN_STACK[4]:='';
END_METHOD

METHOD HOME_RETURN
VAR_INPUT
	ENA: BOOL;
END_VAR
VAR
	TEMP:STRING;
END_VAR
IF ENA = FALSE THEN
	RETURN;
END_IF

IF (DIAGS_OPEN > 0) THEN
	GVL_System.CLOSE_DLGS:=TRUE;
	RETURN;
END_IF

TEMP := POP_RET_STACK();

IF LEN(TEMP) > 0 THEN
	// we have a return page!
	VisuElems.CurrentVisu := TEMP;
ELSE
	VisuElems.CurrentVisu := DEFAULT_HOME_PAGE;
END_IF
END_METHOD

METHOD GOTO_PAGE
VAR_INPUT
	ENA: BOOL;
	NEW_PAGE: STRING;
	RETURN_PAGE: STRING:='';
END_VAR
IF ENA = FALSE THEN
	RETURN;
END_IF

IF LEN(RETURN_PAGE) > 0 THEN
	PUSH_RET_STACK(RETURN_PAGE);
ELSE
	PUSH_RET_STACK(VisuElems.CurrentVisu); 	
END_IF

VisuElems.CurrentVisu := NEW_PAGE;
END_METHOD

METHOD PUSH_RET_STACK
VAR_INPUT
	NEW_PAGE: STRING;
END_VAR
RETURN_STACK[4]:=RETURN_STACK[3];
RETURN_STACK[3]:=RETURN_STACK[2];
RETURN_STACK[2]:=RETURN_STACK[1];
RETURN_STACK[1]:=RETURN_STACK[0];
RETURN_STACK[0]:=NEW_PAGE;
END_METHOD

METHOD POP_RET_STACK : STRING
VAR_INPUT
END_VAR
POP_RET_STACK:=RETURN_STACK[0];
RETURN_STACK[0]:=RETURN_STACK[1];
RETURN_STACK[1]:=RETURN_STACK[2];
RETURN_STACK[2]:=RETURN_STACK[3];
RETURN_STACK[3]:=RETURN_STACK[4];
RETURN_STACK[4]:='';
END_METHOD

END_PROGRAM

// Device/Application/LIBS/HMI/Nav_SetupHalo
PROGRAM Nav_SetupHalo
VAR
	pClient : POINTER TO VisuElems.VisuStructClientData;
	stSelColors: VisuElems.VisuStructColors;
	SelColor_DWORD: DWORD := 16#FF84DE02;
	FrameOffset: INT := -5;
END_VAR

VAR_INPUT
	ENA:BOOL;
END_VAR

IF ENA=FALSE THEN
	RETURN;
END_IF

stSelColors:=VisuElems.g_SelectionManager.SelectionColors;
stSelColors.dwFrameColor:=SelColor_DWORD;
VisuElems.g_SelectionManager.FrameOffset:=FrameOffset;
VisuElems.g_SelectionManager.SelectionColors:=stSelColors;

END_PROGRAM

// Device/Application/LIBS/HMI/CheckDlgsOpen
PROGRAM CheckDlgsOpen
VAR_INPUT
	Names: ARRAY[0..19] OF STRING(40);
END_VAR
VAR
    pstClientData       : POINTER TO VisuElems.VisuStructClientData;
    itfDialogManager    : VisuElems.IDialogManager;
    itfMyDialog         : VisuElems.IVisualisationDialog;
	CheckDialogOpen: BOOL; 
	X: INT;
END_VAR
VAR_OUTPUT
	COUNT: WORD;
END_VAR

VisuElems.g_ClientManager.BeginIteration();

COUNT:=0;

WHILE (pstClientData := VisuElems.VisuElemBase.g_ClientManager.GetNextClient()) <> 0 DO
	FOR X:= 0 TO 19 DO	
		IF (LEN(Names[X])>0) THEN
			itfDialogManager    := VisuElems.g_VisuManager.GetDialogManager();	
			itfMyDialog         := itfDialogManager.GetDialog(Names[X]);	
			CheckDialogOpen     := VisuDialogs.VisuDlgUtil_IsDialogOpen(itfMyDialog,pstClientData,itfDialogManager);
	
			IF CheckDialogOpen THEN
				COUNT:=COUNT+1;
			END_IF
		END_IF					
	END_FOR
END_WHILE

END_PROGRAM

// Device/Application/LIBS/HMI/CloseDlgs
PROGRAM CloseDlgs
VAR
	pstClientData: POINTER TO VisuElems.VisuStructClientData;
	itfDialogManager: VisuElems.IDialogManager;
END_VAR
VAR_OUTPUT
	COUNT: WORD;
END_VAR

VisuElems.VisuElemBase.g_ClientManager.BeginIteration();
pstClientData:= VisuElems.VisuElemBase.g_ClientManager.GetNextClient();

WHILE pstClientData <> 0 DO
	itfDialogManager := VisuElems.g_VisuManager.GetDialogManager();
	itfDialogManager.CloseAllOpenDialogs(pstClientData);
	pstClientData:= VisuElems.VisuElemBase.g_ClientManager.GetNextClient();
END_WHILE

END_PROGRAM

// Device/Application/LIBS/HMI/Nav_Get_Page_Name
PROGRAM Nav_Get_Page_Name
VAR_INPUT
	ENA:BOOL;
	VIZNAME_Prefix: STRING;
END_VAR

VAR_OUTPUT
	Head_PageName: STRING;
END_VAR

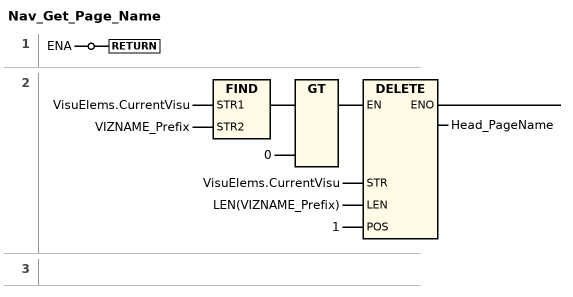
// NETWORK 1
IF NOT ENA THEN RETURN; END_IF

// NETWORK 2
IF FIND(STR1 := VisuElems.CurrentVisu, STR2 := VIZNAME_Prefix) > 0 THEN
    Head_PageName := DELETE(STR := VisuElems.CurrentVisu, LEN := LEN(VIZNAME_Prefix), POS := 1);
END_IF

// NETWORK 3

END_PROGRAM

// Device/Application/LIBS/HMI/Nav_Pages_Group_FB
FUNCTION_BLOCK Nav_Pages_Group_FB
VAR
	Index_Update:BOOL;
	iCounter: INT;
	PageActiveIndex:INT:=0;	
END_VAR

VAR_INPUT
	EnterFirstPage:BOOL;
	EnterSelectedPage:BOOL;
	EnterSelectedIndex:INT;
	Names: ARRAY[0..19] OF STRING(40);
	NumPages: INT;
	Nav_Left: BOOL;
	Nav_Right: BOOL;
	LoopBackLastPage:BOOL;
	DIAGS_OPEN: BOOL;
END_VAR

VAR_OUTPUT
	Active:BOOL;
	Page_Index:INT;
	ShowNavLeftIcon:BOOL;
	ShowNavRightIcon:BOOL;
END_VAR

VAR_IN_OUT
	CurrentVisu: STRING;
END_VAR

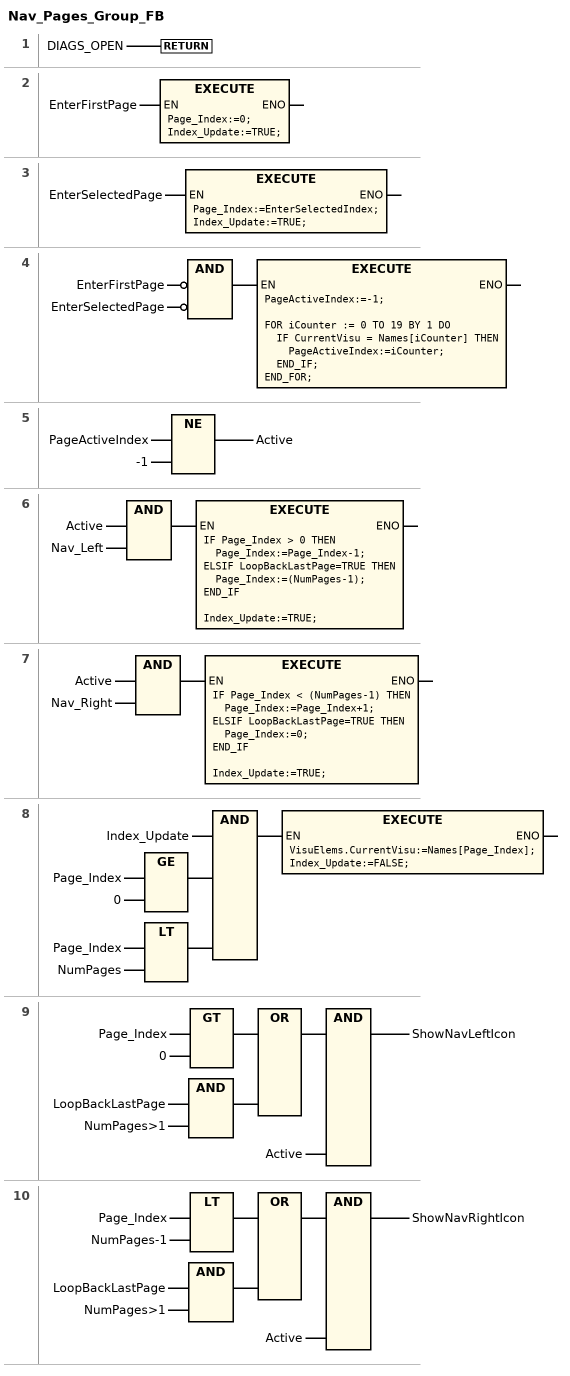
// NETWORK 1
IF DIAGS_OPEN THEN RETURN; END_IF

// NETWORK 2
IF EnterFirstPage THEN
    Page_Index:=0;
    Index_Update:=TRUE;
END_IF

// NETWORK 3
IF EnterSelectedPage THEN
    Page_Index:=EnterSelectedIndex;
    Index_Update:=TRUE;
END_IF

// NETWORK 4
IF NOT EnterFirstPage AND NOT EnterSelectedPage THEN
    PageActiveIndex:=-1;
    
    FOR iCounter := 0 TO 19 BY 1 DO
    	IF CurrentVisu = Names[iCounter] THEN
    		PageActiveIndex:=iCounter;
    	END_IF;
    END_FOR;
END_IF

// NETWORK 5
Active := PageActiveIndex <> -1;

// NETWORK 6
IF Active AND Nav_Left THEN
    IF Page_Index > 0 THEN
    	Page_Index:=Page_Index-1;
    ELSIF LoopBackLastPage=TRUE THEN
    	Page_Index:=(NumPages-1);
    END_IF
    
    Index_Update:=TRUE;
END_IF

// NETWORK 7
IF Active AND Nav_Right THEN
    IF Page_Index < (NumPages-1) THEN
    	Page_Index:=Page_Index+1;
    ELSIF LoopBackLastPage=TRUE THEN
    	Page_Index:=0;
    END_IF
    
    Index_Update:=TRUE;
END_IF

// NETWORK 8
IF Index_Update AND Page_Index >= 0 AND Page_Index < NumPages THEN
    VisuElems.CurrentVisu:=Names[Page_Index];
    Index_Update:=FALSE;
END_IF

// NETWORK 9
ShowNavLeftIcon := (Page_Index > 0 OR LoopBackLastPage AND (NumPages>1)) AND Active;

// NETWORK 10
ShowNavRightIcon := (Page_Index < (NumPages-1) OR LoopBackLastPage AND (NumPages>1)) AND Active;

END_FUNCTION_BLOCK

// Device/Application/App_Common/System/PLC_SYSTEM
PROGRAM PLC_SYSTEM
VAR
	INIT: BOOL:=TRUE;
	
	Epcoh_Update_TON: TON;
	
	MacAsString: STRING(1024);
	MacAsStringResult: INT;	
	
	Cycle_Freq_FB: Cycle_Freq_REAL;	
	
	SystemUpTimeMs: DWORD;
	SystemCyclesFreq: REAL;
	
	System_Battery_V: REAL;
	SIM_System_mV: BOOL;
	Battery_Warning_TON: TON;
	Battery_Warning_Reset_TON: TON;
	
	CHASSIS_UDP_Info_Viz: UDP_Info_Viz;
	
	TickMs: UDINT;
	TickMsWarmInit: UDINT;
	
	Date_and_time_format: STRING(30);
	
	TimeEpochAsUDINT: UDINT;
	TimeEpochAsString: STRING;
	DisplayDateTimeString: STRING;
	
	Reset_Settings: BOOL;
	Reset_Settings_Applied: BOOL;
	Reset_Settings_TON: TON;
	Reset_Settings_Applied_TOF: TOF;
END_VAR
VAR // added by the converter: edge detectors and wires of the graphical bodies
    _rt1 : R_TRIG;
END_VAR

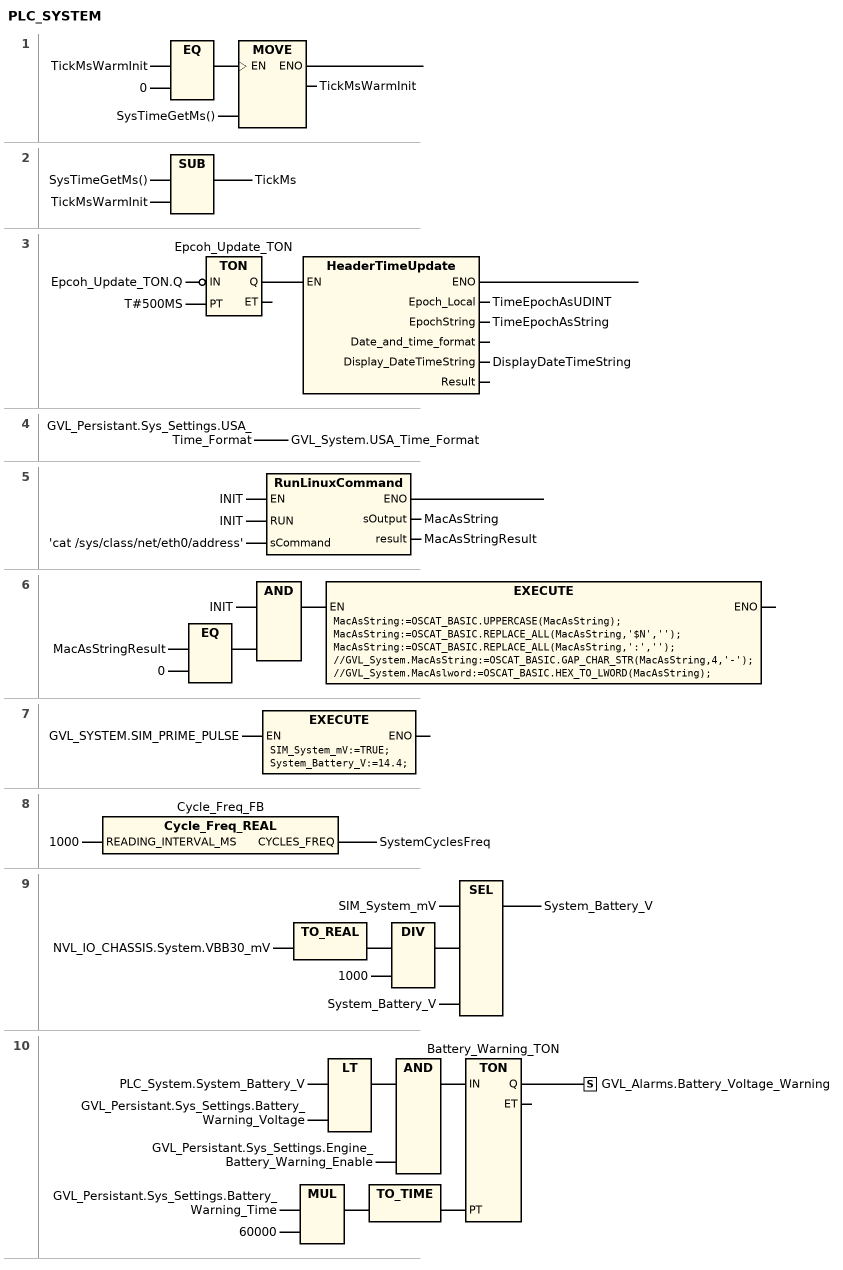
// NETWORK 1
_rt1(CLK := TickMsWarmInit = 0);
IF _rt1.Q THEN TickMsWarmInit := SysTimeGetMs(); END_IF

// NETWORK 2
TickMs := (SysTimeGetMs()) - TickMsWarmInit;

// NETWORK 3
Epcoh_Update_TON(IN := NOT Epcoh_Update_TON.Q, PT := T#500MS); // TON
IF Epcoh_Update_TON.Q THEN
    HeaderTimeUpdate(Epoch_Local => TimeEpochAsUDINT, EpochString => TimeEpochAsString, Display_DateTimeString => DisplayDateTimeString);
END_IF

// NETWORK 4
GVL_System.USA_Time_Format := GVL_Persistant.Sys_Settings.USA_Time_Format;

// NETWORK 5
IF INIT THEN
    RunLinuxCommand(RUN := INIT, sCommand := 'cat /sys/class/net/eth0/address', sOutput => MacAsString, result => MacAsStringResult);
END_IF

// NETWORK 6
IF INIT AND MacAsStringResult = 0 THEN
    MacAsString:=OSCAT_BASIC.UPPERCASE(MacAsString);
    MacAsString:=OSCAT_BASIC.REPLACE_ALL(MacAsString,'$N','');
    MacAsString:=OSCAT_BASIC.REPLACE_ALL(MacAsString,':','');
    //GVL_System.MacAsString:=OSCAT_BASIC.GAP_CHAR_STR(MacAsString,4,'-');
    //GVL_System.MacAslword:=OSCAT_BASIC.HEX_TO_LWORD(MacAsString);
END_IF

// NETWORK 7
IF GVL_SYSTEM.SIM_PRIME_PULSE THEN
    SIM_System_mV:=TRUE;
    System_Battery_V:=14.4;
END_IF

// NETWORK 8
Cycle_Freq_FB(READING_INTERVAL_MS := 1000); // Cycle_Freq_REAL
SystemCyclesFreq := Cycle_Freq_FB.CYCLES_FREQ;

// NETWORK 9
System_Battery_V := SEL(SIM_System_mV, TO_REAL(NVL_IO_CHASSIS.System.VBB30_mV) / 1000, System_Battery_V);

// NETWORK 10
Battery_Warning_TON(IN := PLC_System.System_Battery_V < GVL_Persistant.Sys_Settings.Battery_Warning_Voltage AND GVL_Persistant.Sys_Settings.Engine_Battery_Warning_Enable, PT := TO_TIME(GVL_Persistant.Sys_Settings.Battery_Warning_Time * 60000)); // TON
GVL_Alarms.Battery_Voltage_Warning S= Battery_Warning_TON.Q;

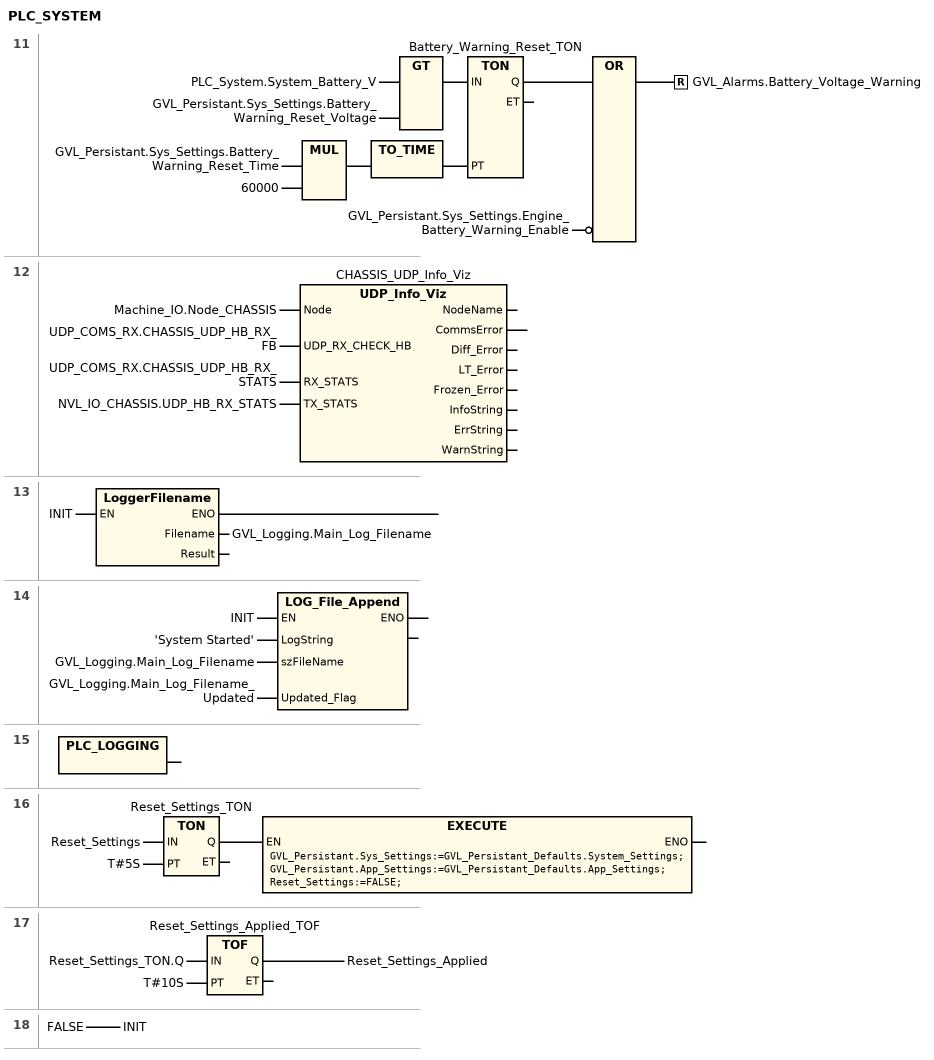
// NETWORK 11
Battery_Warning_Reset_TON(IN := PLC_System.System_Battery_V > GVL_Persistant.Sys_Settings.Battery_Warning_Reset_Voltage, PT := TO_TIME(GVL_Persistant.Sys_Settings.Battery_Warning_Reset_Time * 60000)); // TON
GVL_Alarms.Battery_Voltage_Warning R= Battery_Warning_Reset_TON.Q OR NOT GVL_Persistant.Sys_Settings.Engine_Battery_Warning_Enable;

// NETWORK 12
CHASSIS_UDP_Info_Viz(
    Node := Machine_IO.Node_CHASSIS,
    UDP_RX_CHECK_HB := UDP_COMS_RX.CHASSIS_UDP_HB_RX_FB,
    RX_STATS := UDP_COMS_RX.CHASSIS_UDP_HB_RX_STATS,
    TX_STATS := NVL_IO_CHASSIS.UDP_HB_RX_STATS); // UDP_Info_Viz

// NETWORK 13
IF INIT THEN LoggerFilename(Filename => GVL_Logging.Main_Log_Filename); END_IF

// NETWORK 14
IF INIT THEN
    LOG_File_Append(LogString := 'System Started', szFileName := GVL_Logging.Main_Log_Filename, Updated_Flag := GVL_Logging.Main_Log_Filename_Updated);
END_IF

// NETWORK 15
PLC_LOGGING();

// NETWORK 16
Reset_Settings_TON(IN := Reset_Settings, PT := T#5S); // TON
IF Reset_Settings_TON.Q THEN
    GVL_Persistant.Sys_Settings:=GVL_Persistant_Defaults.System_Settings;
    GVL_Persistant.App_Settings:=GVL_Persistant_Defaults.App_Settings;
    Reset_Settings:=FALSE;
END_IF

// NETWORK 17
Reset_Settings_Applied_TOF(IN := Reset_Settings_TON.Q, PT := T#10S); // TOF
Reset_Settings_Applied := Reset_Settings_Applied_TOF.Q;

// NETWORK 18
INIT := FALSE;

METHOD LoggerFilename

VAR
	Date_and_time_in_seconds : UDINT;
	Date_and_Time_result : UDINT;
	Epoch_Local : UDINT;	
	Date_and_time_format: DT;
END_VAR

VAR_IN_OUT
END_VAR

VAR_OUTPUT
	Filename : STRING:='Log_Deault.txt';
	Result: INT;
END_VAR
// Get time in seconds since 1970 :
Date_and_time_in_seconds := SysTimeRtc.SysTimeRtcGet(Date_and_Time_result);
IF Date_and_Time_result <> 0 THEN
	Result:=-1;
	RETURN;
END_IF

// Convert UTC seconds to local time seconds, regarding Timezone and Summer time :
Date_and_Time_result := SysTimeRtc.SysTimeRtcConvertUtcToLocal(Date_and_time_in_seconds, Epoch_Local);
IF Date_and_Time_result <> 0 THEN
	Result:=-2;	
	RETURN;
END_IF

Filename:='AppLogs/Log_';
Filename:= CONCAT(Filename,OSCAT_BASIC.DT_TO_STRF(DTI:=TO_DT(Epoch_Local), MS:=0, FMT:='#D#H#A',LANG:=OSCAT_BASIC.language.DEFAULT));
Filename:= CONCAT(Filename,'.txt');
Result:=0;
END_METHOD

METHOD HeaderTimeUpdate

VAR
	Date_and_time_in_seconds : UDINT;
	Date_and_Time_result : UDINT;
	Local_date_time_from_secs : SYSTIMEDATE;	
END_VAR

VAR_IN_OUT
END_VAR

VAR_OUTPUT
	Epoch_Local : UDINT;
	EpochString: STRING;	
	Date_and_time_format: DT;
	Display_DateTimeString : STRING;
	Result:INT;
END_VAR
// Get time in seconds since 1970 :
Date_and_time_in_seconds := SysTimeRtc.SysTimeRtcGet(Date_and_Time_result);
IF Date_and_Time_result <> 0 THEN
	Result:=-1;
	RETURN;
END_IF

// Convert UTC seconds to local time seconds, regarding Timezone and Summer time :
Date_and_Time_result := SysTimeRtc.SysTimeRtcConvertUtcToLocal(Date_and_time_in_seconds, Epoch_Local);
IF Date_and_Time_result <> 0 THEN
	Result:=-2;	
	RETURN;
END_IF

//EpochString:=OSCAT_BASIC.DWORD_TO_STRING_LEADING_ZEROS(Epoch_Local,12);
//EpochString:=OSCAT_BASIC.GAP_CHAR_STR(EpochString,4,' ');

// Convert DATE_AND_TIME to a String :
IF GVL_Persistant.Sys_Settings.USA_Time_Format THEN
	Display_DateTimeString:= OSCAT_BASIC.DT_TO_STRF(DTI:=TO_DT(Epoch_Local), MS:=0, FMT:='#D-#H-#A #N:#R:#T',LANG:=OSCAT_BASIC.language.DEFAULT);
ELSE
	Display_DateTimeString:= OSCAT_BASIC.DT_TO_STRF(DTI:=TO_DT(Epoch_Local), MS:=0, FMT:='#H-#D-#A #N:#R:#T',LANG:=OSCAT_BASIC.language.DEFAULT);
END_IF

Result:=0;
END_METHOD

END_PROGRAM

// Device/Application/LIBS/HMI/RunLinuxCommand
PROGRAM RunLinuxCommand
VAR_INPUT
	RUN: BOOL;
	sCommand : STRING(1024);
END_VAR

VAR_OUTPUT
	sOutput : STRING(1024);
	result : INT;	
END_VAR

VAR
	refCommand : REFERENCE TO STRING(1024);
	refOutput : REFERENCE TO STRING(1024);
END_VAR

VAR_IN_OUT
END_VAR

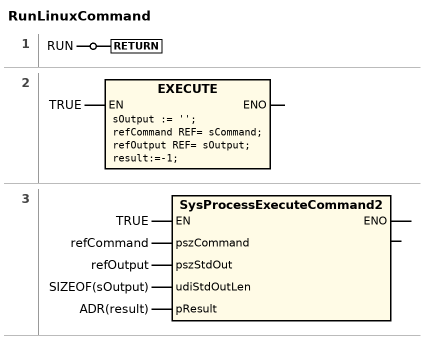
// NETWORK 1
IF NOT RUN THEN RETURN; END_IF

// NETWORK 2
sOutput := '';
refCommand REF= sCommand;
refOutput REF= sOutput;
result:=-1;

// NETWORK 3
SysProcessExecuteCommand2(pszCommand := refCommand, pszStdOut := refOutput, udiStdOutLen := SIZEOF(sOutput), pResult := ADR(result));

END_PROGRAM

// Device/Application/LIBS/UDP/UDP_Info_Viz
FUNCTION_BLOCK UDP_Info_Viz
VAR_INPUT
	Node: REFERENCE TO NodeComFB;
	UDP_RX_CHECK_HB: REFERENCE TO UDP_RX_CHECK_HB_FB;
	RX_STATS: REFERENCE TO UDP_RX_STATS_HB_STRUCT;
	TX_STATS: REFERENCE TO UDP_RX_STATS_HB_STRUCT;
END_VAR
VAR
	TempString: STRING(1024);	
END_VAR

VAR_OUTPUT
	NodeName: STRING;
	CommsError:BOOL;
	Diff_Error:BOOL;
	LT_Error:BOOL;
	Frozen_Error:BOOL;
	InfoString: STRING(1024);
	ErrString: STRING(1024);
	WarnString: STRING(1024);	
END_VAR

IF __ISVALIDREF(Node)=FALSE THEN
	RETURN;
END_IF

IF __ISVALIDREF(UDP_RX_CHECK_HB)=FALSE THEN
	RETURN;
END_IF

IF __ISVALIDREF(RX_STATS)=FALSE THEN
	RETURN;
END_IF

IF __ISVALIDREF(TX_STATS)=FALSE THEN
	RETURN;
END_IF

TempString:= '';
TempString:=CONCAT(TempString,print_formated_DINT_func('RX_PLC_UpTimeMs:      ','%6d',RX_STATS.PLC_UpTimeMs));
TempString:=CONCAT(TempString,'$0d');
TempString:=CONCAT(TempString,print_formated_DINT_func('RX_PLC_UpTimeMs_Diff: ','%6d',RX_STATS.PLC_UpTimeMs_Diff));
TempString:=CONCAT(TempString,'$0d');
TempString:=CONCAT(TempString,print_formated_DINT_func('RX_PLC_UpTimeMs_Last: ','%6d',RX_STATS.PLC_UpTimeMs_Last));
TempString:=CONCAT(TempString,'$0d');

TempString:=CONCAT(TempString,print_formated_DINT_func('TX_PLC_UpTimeMs:      ','%6d',TX_STATS.PLC_UpTimeMs));
TempString:=CONCAT(TempString,'$0d');
TempString:=CONCAT(TempString,print_formated_DINT_func('TX_PLC_UpTimeMs_Diff: ','%6d',TX_STATS.PLC_UpTimeMs_Diff));
TempString:=CONCAT(TempString,'$0d');
TempString:=CONCAT(TempString,print_formated_DINT_func('TX_PLC_UpTimeMs_Last: ','%6d',TX_STATS.PLC_UpTimeMs_Last));

InfoString:=TempString;

TempString:= '';
TempString:=CONCAT(TempString,print_formated_DINT_func('RX_Err_LT:    ','%4d',RX_STATS.Error_LT_Count));
TempString:=CONCAT(TempString,'$0d');
TempString:=CONCAT(TempString,print_formated_DINT_func('RX_Err_Diff:  ','%4d',RX_STATS.Error_Diff_Count));
TempString:=CONCAT(TempString,'$0d');
TempString:=CONCAT(TempString,print_formated_DINT_func('RX_Err_Frozen:','%4d',RX_STATS.Error_Frozen_Count));
TempString:=CONCAT(TempString,'$0d');
TempString:=CONCAT(TempString,print_formated_DINT_func('TX_Err_LT:    ','%4d',TX_STATS.Error_LT_Count));
TempString:=CONCAT(TempString,'$0d');
TempString:=CONCAT(TempString,print_formated_DINT_func('TX_Err_Diff:  ','%4d',TX_STATS.Error_Diff_Count));
TempString:=CONCAT(TempString,'$0d');
TempString:=CONCAT(TempString,print_formated_DINT_func('TX_Err_Frozen:','%4d',TX_STATS.Error_Frozen_Count));

ErrString:=TempString;

TempString:= '';
TempString:=CONCAT(TempString,print_formated_DINT_func('RX_Warn_LT:     ','%4d',RX_STATS.Warn_LT_Count));
TempString:=CONCAT(TempString,'$0d');
TempString:=CONCAT(TempString,print_formated_DINT_func('RX_Warn_Diff:   ','%4d',RX_STATS.Warn_Diff_Count));
TempString:=CONCAT(TempString,'$0d');
TempString:=CONCAT(TempString,print_formated_DINT_func('RX_Warn_Frozen:','%4d',RX_STATS.Warn_Frozen_Count));
TempString:=CONCAT(TempString,'$0d');
TempString:=CONCAT(TempString,print_formated_DINT_func('TX_Warn_LT:     ','%4d',TX_STATS.Warn_LT_Count));
TempString:=CONCAT(TempString,'$0d');
TempString:=CONCAT(TempString,print_formated_DINT_func('TX_Warn_Diff:   ','%4d',TX_STATS.Warn_Diff_Count));
TempString:=CONCAT(TempString,'$0d');
TempString:=CONCAT(TempString,print_formated_DINT_func('TX_Warn_Frozen:','%4d',TX_STATS.Warn_Frozen_Count));

WarnString:=TempString;

NodeName:= Node.Full_Name;
CommsError:= UDP_RX_CHECK_HB.CommsError;
Diff_Error:= UDP_RX_CHECK_HB.Error_Diff;
LT_Error:=UDP_RX_CHECK_HB.Error_LessThan;
Frozen_Error:=UDP_RX_CHECK_HB.Error_Frozen;

END_FUNCTION_BLOCK

// Device/Application/LIBS/print_formated_DINT_func
FUNCTION print_formated_DINT_func : STRING
VAR_INPUT
	Prefix: STRING;
	FormatString: STRING:='%.1fHz';
	Value:DINT;	
END_VAR
VAR
	TempString: STRING;
END_VAR

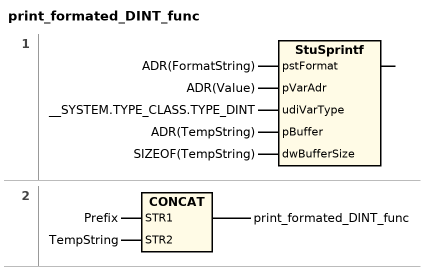
// NETWORK 1
StuSprintf(pstFormat := ADR(FormatString), pVarAdr := ADR(Value), udiVarType := __SYSTEM.TYPE_CLASS.TYPE_DINT, pBuffer := ADR(TempString), dwBufferSize := SIZEOF(TempString));

// NETWORK 2
print_formated_DINT_func := CONCAT(STR1 := Prefix, STR2 := TempString);

END_FUNCTION

// Device/Application/LIBS/IO Common/NodeComFB
FUNCTION_BLOCK NodeComFB
VAR_INPUT
	Full_Name: STRING;
	Short_Name: STRING;
	Unavail:BOOL;
	Fault: BOOL;
	Warn: BOOL;	
END_VAR
VAR_OUTPUT
END_VAR
VAR
END_VAR

END_FUNCTION_BLOCK

// Device/Application/App_Common/UDP/UDP_COMS_RX
PROGRAM UDP_COMS_RX
VAR
	CYCLE_FREQ_FB_0: SLL_Common.Cycle_Freq;
	TIMESTAMP_TO_FB_0: SLL_Common.Timestamp_TO;

	CHASSIS_UDP_HB_RX_FB: UDP_RX_CHECK_HB_FB;
	
	CHASSIS_UDP_HB_RX_STATS: UDP_RX_STATS_HB_STRUCT;	
	
	RESET_COMMS_ERROR: BOOL;
	UDP_RX_WAIT_CHECK_TON: TON;
	UDP_RX_WAIT_CHECK_TEST: BOOL;

	UDP_RX_MONITORING_MS: DINT :=4000;
	UDP_RX_WARNING_DIFF_THRESHOLD: DINT := 400;
	UDP_RX_ERROR_DIFF_THRESHOLD: DINT := 500;
	UDP_RX_WARNING_FROZEN_THRESHOLD: DINT := 400;
	UDP_RX_ERROR_FROZEN_THRESHOLD: DINT :=500;
	UDP_RX_ERROR_MISSING_MS: DINT :=500;
	UDP_RX_ERROR_RECOVERY_MS: DINT :=3000;
	
	RESET_ETHERNET_COMMS_TP: TP;
	RESET_ETHERNET_COMMS_AUTO: BOOL;
	RESET_ETHERNET_COMMS_TON: TON;
	RESET_STATS: BOOL;
	
	RESET_ALARMS: BOOL;	
	RESET_ETHERNET_COMMS_AUTO_ENA: BOOL := FALSE;
	
	CHASSIS_PLC_RED_CROSS: BOOL;
END_VAR
VAR // added by the converter: edge detectors and wires of the graphical bodies
    _w1 : BOOL;
END_VAR

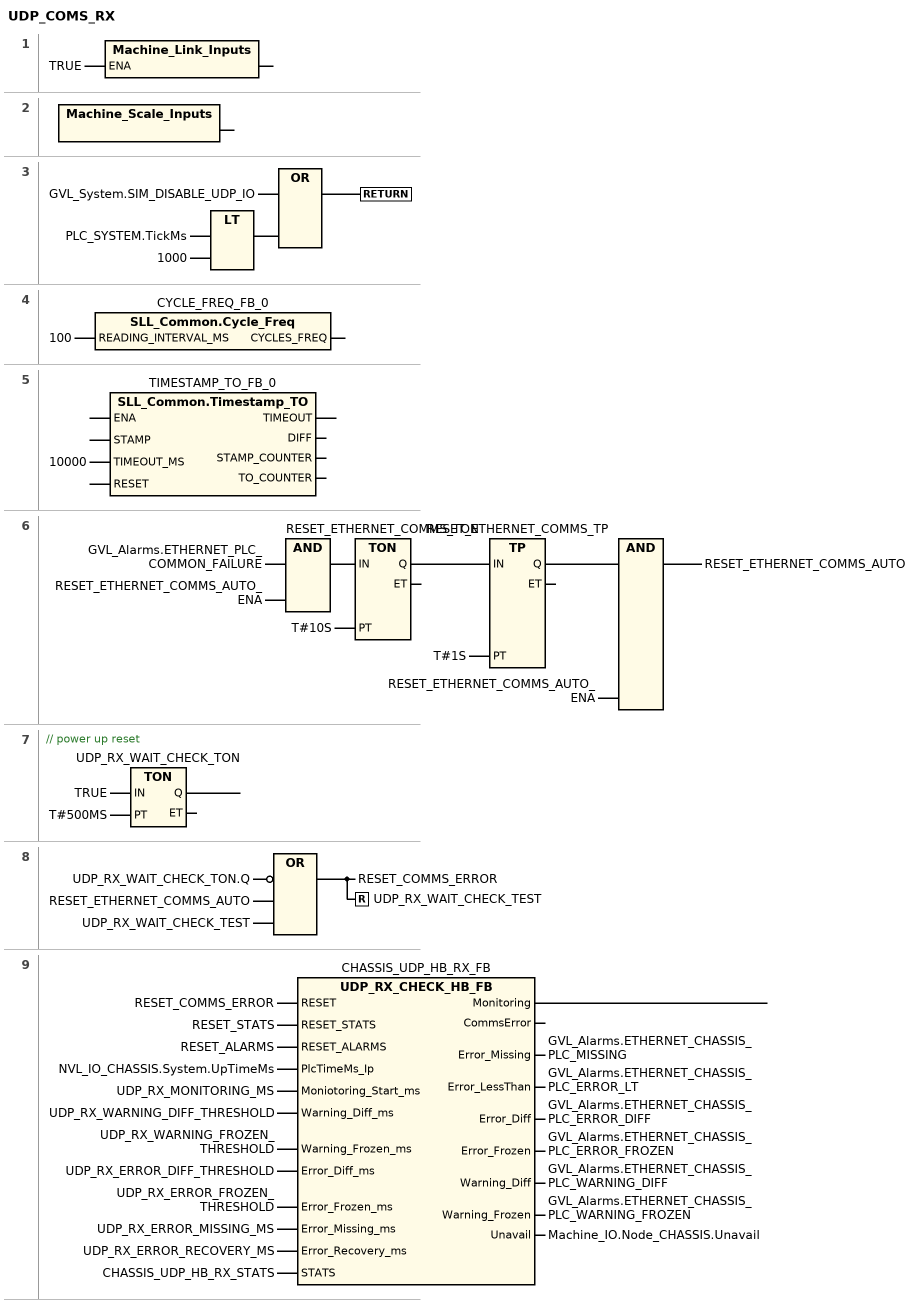
// NETWORK 1
Machine_Link_Inputs(ENA := TRUE);

// NETWORK 2
Machine_Scale_Inputs();

// NETWORK 3
IF GVL_System.SIM_DISABLE_UDP_IO OR PLC_SYSTEM.TickMs < 1000 THEN RETURN; END_IF

// NETWORK 4
CYCLE_FREQ_FB_0(READING_INTERVAL_MS := 100); // SLL_Common.Cycle_Freq

// NETWORK 5
TIMESTAMP_TO_FB_0(TIMEOUT_MS := 10000); // SLL_Common.Timestamp_TO

// NETWORK 6
RESET_ETHERNET_COMMS_TON(IN := GVL_Alarms.ETHERNET_PLC_COMMON_FAILURE AND RESET_ETHERNET_COMMS_AUTO_ENA, PT := T#10S); // TON
RESET_ETHERNET_COMMS_TP(IN := RESET_ETHERNET_COMMS_TON.Q, PT := T#1S); // TP
RESET_ETHERNET_COMMS_AUTO := RESET_ETHERNET_COMMS_TP.Q AND RESET_ETHERNET_COMMS_AUTO_ENA;

// NETWORK 7
// // power up reset
UDP_RX_WAIT_CHECK_TON(IN := TRUE, PT := T#500MS); // TON

// NETWORK 8
_w1 := NOT UDP_RX_WAIT_CHECK_TON.Q OR RESET_ETHERNET_COMMS_AUTO OR UDP_RX_WAIT_CHECK_TEST;
RESET_COMMS_ERROR := _w1;
UDP_RX_WAIT_CHECK_TEST R= _w1;

// NETWORK 9
CHASSIS_UDP_HB_RX_FB(
    RESET := RESET_COMMS_ERROR,
    RESET_STATS := RESET_STATS,
    RESET_ALARMS := RESET_ALARMS,
    PlcTimeMs_Ip := NVL_IO_CHASSIS.System.UpTimeMs,
    Moniotoring_Start_ms := UDP_RX_MONITORING_MS,
    Warning_Diff_ms := UDP_RX_WARNING_DIFF_THRESHOLD,
    Warning_Frozen_ms := UDP_RX_WARNING_FROZEN_THRESHOLD,
    Error_Diff_ms := UDP_RX_ERROR_DIFF_THRESHOLD,
    Error_Frozen_ms := UDP_RX_ERROR_FROZEN_THRESHOLD,
    Error_Missing_ms := UDP_RX_ERROR_MISSING_MS,
    Error_Recovery_ms := UDP_RX_ERROR_RECOVERY_MS,
    STATS := CHASSIS_UDP_HB_RX_STATS,
    Error_Missing => GVL_Alarms.ETHERNET_CHASSIS_PLC_MISSING,
    Error_LessThan => GVL_Alarms.ETHERNET_CHASSIS_PLC_ERROR_LT,
    Error_Diff => GVL_Alarms.ETHERNET_CHASSIS_PLC_ERROR_DIFF,
    Error_Frozen => GVL_Alarms.ETHERNET_CHASSIS_PLC_ERROR_FROZEN,
    Warning_Diff => GVL_Alarms.ETHERNET_CHASSIS_PLC_WARNING_DIFF,
    Warning_Frozen => GVL_Alarms.ETHERNET_CHASSIS_PLC_WARNING_FROZEN,
    Unavail => Machine_IO.Node_CHASSIS.Unavail); // UDP_RX_CHECK_HB_FB

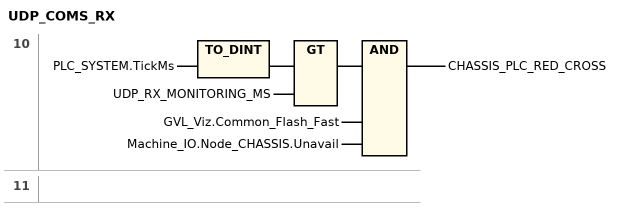
// NETWORK 10
CHASSIS_PLC_RED_CROSS := TO_DINT(PLC_SYSTEM.TickMs) > UDP_RX_MONITORING_MS AND GVL_Viz.Common_Flash_Fast AND Machine_IO.Node_CHASSIS.Unavail;

// NETWORK 11

END_PROGRAM

// Device/Application/App_CODE_GEN/MAIN_CODE_GEN/App_CODE_GEN/Machine IO/Funcs/Machine_Link_Inputs
PROGRAM Machine_Link_Inputs
VAR_INPUT
	ENA:BOOL;
END_VAR

VAR
	INIT_ONCE:BOOL:=TRUE;
	Init_Input_Links:BOOL :=TRUE;
END_VAR

IF Init_Input_Links THEN
	Machine_Link_Inputs_Init();	
	Init_Input_Links:=FALSE;
END_IF

// Machine_Link_Inputs_Main_CODE_GEN_START

// generated (UTC): 2024-07-23 18:31:25.048386+00:00

Machine_IO.Inputs.ESTOP_OK(); // CR0709.IN0100
Machine_IO.Inputs.DRUM_PRESSURE(); // CR0709.IN0101
Machine_IO.Inputs.Radial_RightLimitSwitch(); // CR0709.IN0102
Machine_IO.Inputs.Radial_LeftLimitSwitch(); // CR0709.IN0103
Machine_IO.Inputs.MachineMode(); // CR0709.IN0200
Machine_IO.Inputs.KeySwitchCranking(); // CR0709.IN0201
Machine_IO.Inputs.SPARE_IN0202(); // CR0709.IN0202
Machine_IO.Inputs.SPARE_IN0203(); // CR0709.IN0203
Machine_IO.Inputs.SPARE_IN0600(); // CR0709.IN0600
Machine_IO.Inputs.SPARE_IN0601(); // CR0709.IN0601
Machine_IO.Inputs.SPARE_IN0602(); // CR0709.IN0602
Machine_IO.Inputs.SPARE_IN0603(); // CR0709.IN0603
Machine_IO.Inputs.SPARE_IN0700(); // CR0709.IN0700
Machine_IO.Inputs.RADIORHS_JACKLEGRAISE_REQ(); // CR0709.IN0701
Machine_IO.Inputs.RHS_TROMMELDOORSW(); // CR0709.IN0702
Machine_IO.Inputs.LHS_TROMMELDOORSW(); // CR0709.IN0703
Machine_IO.Inputs.HYDOILTEMP_SW(); // CR0709.IN0000
Machine_IO.Inputs.HYDOILLEVEL_SW(); // CR0709.IN0001
Machine_IO.Inputs.THERMOSTAT(); // CR0709.IN0002
Machine_IO.Inputs.RADIORHS_JACKLEGLOWER_REQ(); // CR0709.IN0003
Machine_IO.Inputs.RADIOLHS_JACKLEGRAISE_REQ(); // CR0709.IN0500
Machine_IO.Inputs.RADIOLHS_JACKLEGLOWER_REQ(); // CR0709.IN0501
Machine_IO.Inputs.SideConvRaise_RadialMoveRight(); // CR0709.IN0502
Machine_IO.Inputs.SideConvLower_RadialMoveLeft(); // CR0709.IN0503
Machine_IO.Inputs.SPARE_IN0400(); // CR0709.IN0400
Machine_IO.Inputs.FUELLEVEL_PERCENT(); // CR0709.IN0401
Machine_IO.Inputs.UMBTRACKREQ(); // CR0709.IN0900
Machine_IO.Inputs.UMBMACHINESTOP(); // CR0709.IN0901
Machine_IO.Inputs.RTF_REQ(); // CR0709.IN0300
Machine_IO.Inputs.RTR_REQ(); // CR0709.IN0301
Machine_IO.Inputs.LTF_REQ(); // CR0709.IN0800
Machine_IO.Inputs.LTR_REQ(); // CR0709.IN0801


// Machine_Link_Inputs_Main_CODE_GEN_STOP

END_PROGRAM

// Device/Application/App_CODE_GEN/MAIN_CODE_GEN/App_CODE_GEN/Machine IO/Funcs/Machine_Link_Inputs_Init
PROGRAM Machine_Link_Inputs_Init
VAR
END_VAR


// Machine_Link_Inputs_Init_CODE_GEN_START

// generated (UTC): 2024-07-23 18:31:25.086388+00:00
Machine_IO.Inputs.ESTOP_OK.Init('CHASSIS','ESTOP_OK','IN0100','a63',NVL_IO_CHASSIS.All_Inputs.IN0100,Machine_IO.Node_CHASSIS);
Machine_IO.Inputs.DRUM_PRESSURE.Init('CHASSIS','DRUM_PRESSURE','IN0101','a64',NVL_IO_CHASSIS.All_Inputs.IN0101,Machine_IO.Node_CHASSIS);
Machine_IO.Inputs.Radial_RightLimitSwitch.Init('CHASSIS','RADIAL_RIGHTLIMIT','IN0102','a65',NVL_IO_CHASSIS.All_Inputs.IN0102,Machine_IO.Node_CHASSIS);
Machine_IO.Inputs.Radial_LeftLimitSwitch.Init('CHASSIS','RADIAL_LEFTLIMIT','IN0103','a66',NVL_IO_CHASSIS.All_Inputs.IN0103,Machine_IO.Node_CHASSIS);
Machine_IO.Inputs.MachineMode.Init('CHASSIS','MACHINE_MODE','IN0200','a67',NVL_IO_CHASSIS.All_Inputs.IN0200,Machine_IO.Node_CHASSIS);
Machine_IO.Inputs.KeySwitchCranking.Init('CHASSIS','KEYSWITCH_CRANKING','IN0201','a68',NVL_IO_CHASSIS.All_Inputs.IN0201,Machine_IO.Node_CHASSIS);
Machine_IO.Inputs.SPARE_IN0202.Init('CHASSIS','SPARE_IN0202','IN0202','a69',NVL_IO_CHASSIS.All_Inputs.IN0202,Machine_IO.Node_CHASSIS);
Machine_IO.Inputs.SPARE_IN0203.Init('CHASSIS','SPARE_IN0203','IN0203','a70',NVL_IO_CHASSIS.All_Inputs.IN0203,Machine_IO.Node_CHASSIS);
Machine_IO.Inputs.SPARE_IN0600.Init('CHASSIS','SPARE_IN0600','IN0600','a55',NVL_IO_CHASSIS.All_Inputs.IN0600,Machine_IO.Node_CHASSIS);
Machine_IO.Inputs.SPARE_IN0601.Init('CHASSIS','SPARE_IN0601','IN0601','a56',NVL_IO_CHASSIS.All_Inputs.IN0601,Machine_IO.Node_CHASSIS);
Machine_IO.Inputs.SPARE_IN0602.Init('CHASSIS','SPARE_IN0602','IN0602','a57',NVL_IO_CHASSIS.All_Inputs.IN0602,Machine_IO.Node_CHASSIS);
Machine_IO.Inputs.SPARE_IN0603.Init('CHASSIS','SPARE_IN0603','IN0603','a58',NVL_IO_CHASSIS.All_Inputs.IN0603,Machine_IO.Node_CHASSIS);
Machine_IO.Inputs.SPARE_IN0700.Init('CHASSIS','SPARE_IN0700','IN0700','a59',NVL_IO_CHASSIS.All_Inputs.IN0700,Machine_IO.Node_CHASSIS);
Machine_IO.Inputs.RADIORHS_JACKLEGRAISE_REQ.Init('CHASSIS','RADIORHS_JACKLEGRAISE_REQ','IN0701','a60',NVL_IO_CHASSIS.All_Inputs.IN0701,Machine_IO.Node_CHASSIS);
Machine_IO.Inputs.RHS_TROMMELDOORSW.Init('CHASSIS','RHS_TROMMELDOORSW','IN0702','a61',NVL_IO_CHASSIS.All_Inputs.IN0702,Machine_IO.Node_CHASSIS);
Machine_IO.Inputs.LHS_TROMMELDOORSW.Init('CHASSIS','LHS_TROMMELDOORSW','IN0703','a62',NVL_IO_CHASSIS.All_Inputs.IN0703,Machine_IO.Node_CHASSIS);
Machine_IO.Inputs.HYDOILTEMP_SW.Init('CHASSIS','HYDOILTEMP_SW','IN0000','a25',NVL_IO_CHASSIS.All_Inputs.IN0000,Machine_IO.Node_CHASSIS);
Machine_IO.Inputs.HYDOILLEVEL_SW.Init('CHASSIS','HYDOILLEVEL_SW','IN0001','a26',NVL_IO_CHASSIS.All_Inputs.IN0001,Machine_IO.Node_CHASSIS);
Machine_IO.Inputs.THERMOSTAT.Init('CHASSIS','THERMOSTAT','IN0002','a27',NVL_IO_CHASSIS.All_Inputs.IN0002,Machine_IO.Node_CHASSIS);
Machine_IO.Inputs.RADIORHS_JACKLEGLOWER_REQ.Init('CHASSIS','RADIORHS_JACKLEGLOWER_REQ','IN0003','a28',NVL_IO_CHASSIS.All_Inputs.IN0003,Machine_IO.Node_CHASSIS);
Machine_IO.Inputs.RADIOLHS_JACKLEGRAISE_REQ.Init('CHASSIS','RADIOLHS_JACKLEGRAISE_REQ','IN0500','a40',NVL_IO_CHASSIS.All_Inputs.IN0500,Machine_IO.Node_CHASSIS);
Machine_IO.Inputs.RADIOLHS_JACKLEGLOWER_REQ.Init('CHASSIS','RADIOLHS_JACKLEGLOWER_REQ','IN0501','a41',NVL_IO_CHASSIS.All_Inputs.IN0501,Machine_IO.Node_CHASSIS);
Machine_IO.Inputs.SideConvRaise_RadialMoveRight.Init('CHASSIS','RADIO_SIDECONVRAISE_RADRIGHT','IN0502','a42',NVL_IO_CHASSIS.All_Inputs.IN0502,Machine_IO.Node_CHASSIS);
Machine_IO.Inputs.SideConvLower_RadialMoveLeft.Init('CHASSIS','RADIO_SIDECONVLOWER_RADLEFT','IN0503','a43',NVL_IO_CHASSIS.All_Inputs.IN0503,Machine_IO.Node_CHASSIS);
Machine_IO.Inputs.SPARE_IN0400.Init('CHASSIS','SPARE_IN0400','IN0400','a46',NVL_IO_CHASSIS.All_Inputs.IN0400,Machine_IO.Node_CHASSIS);
Machine_IO.Inputs.FUELLEVEL_PERCENT.Init('CHASSIS','FUELLEVEL_PERCENT','IN0401','a47',NVL_IO_CHASSIS.All_Inputs.IN0401,Machine_IO.Node_CHASSIS);
Machine_IO.Inputs.UMBTRACKREQ.Init('CHASSIS','UMBTRACKREQ','IN0900','a38',NVL_IO_CHASSIS.All_Inputs.IN0900,Machine_IO.Node_CHASSIS);
Machine_IO.Inputs.UMBMACHINESTOP.Init('CHASSIS','UMBMACHINESTOP','IN0901','a39',NVL_IO_CHASSIS.All_Inputs.IN0901,Machine_IO.Node_CHASSIS);
Machine_IO.Inputs.RTF_REQ.Init('CHASSIS','RTF_REQ','IN0300','a44',NVL_IO_CHASSIS.All_Inputs.IN0300,Machine_IO.Node_CHASSIS);
Machine_IO.Inputs.RTR_REQ.Init('CHASSIS','RTR_REQ','IN0301','a45',NVL_IO_CHASSIS.All_Inputs.IN0301,Machine_IO.Node_CHASSIS);
Machine_IO.Inputs.LTF_REQ.Init('CHASSIS','LTF_REQ','IN0800','a36',NVL_IO_CHASSIS.All_Inputs.IN0800,Machine_IO.Node_CHASSIS);
Machine_IO.Inputs.LTR_REQ.Init('CHASSIS','LTR_REQ','IN0801','a37',NVL_IO_CHASSIS.All_Inputs.IN0801,Machine_IO.Node_CHASSIS);


// Machine_Link_Inputs_Init_CODE_GEN_STOP

END_PROGRAM

// Device/Application/App_CODE_GEN/MAIN_CODE_GEN/App_CODE_GEN/Machine IO/Funcs/Machine_Scale_Inputs
PROGRAM Machine_Scale_Inputs
VAR CONSTANT
END_VAR

VAR
	Scale_DRUM_PRESSURE: pil.ScaleBlock;
	Smooth_DRUM_PRESSURE: fbSmoothing;
	Scale_FUEL_LEVEL: pil.ScaleBlock;
	Smooth_FUEL_LEVEL: fbSmoothing;
END_VAR

